    (* One configurator per IPM state (OUT + 4 targets). Writes the
       per-state sName and fDelta. Ticked cyclically in the body AFTER
       fbStates so its writes win over the template baseline
       FB_StateSetup applied via FB_CC_StatePMPSConfig. Idempotent once
       stPositionState.bUpdated trips. *)
    afbStateDefaults : ARRAY[1..5] OF FB_CC_InternalStateConfig[
        (stPositionState := astPositionState[1][E_IPM_States.OUT],
         sName           := 'OUT',
         fDelta          := FDELTA_DEFAULT),
        (stPositionState := astPositionState[1][E_IPM_States.TARGET1],
         sName           := 'TARGET1',
         fDelta          := FDELTA_DEFAULT),
        (stPositionState := astPositionState[1][E_IPM_States.TARGET2],
         sName           := 'TARGET2',
         fDelta          := FDELTA_DEFAULT),
        (stPositionState := astPositionState[1][E_IPM_States.TARGET3],
         sName           := 'TARGET3',
         fDelta          := FDELTA_DEFAULT),
        (stPositionState := astPositionState[1][E_IPM_States.TARGET4],
         sName           := 'TARGET4',
         fDelta          := FDELTA_DEFAULT)
    ];

    {attribute 'pytmc' := 'pv: MMS'}
    fbStates : FB_PositionStatePMPSND(
        aiMotionStage         := aiMotionStage,
        astPositionState      := astPositionState,
        nActiveMotorCount     := 1,
        eEnumSet              := eEnumSet,
        eEnumGet              := eEnumGet,
        bEnableMotion         := bEnableMotion,
        eMotionRequestPolicy  := E_MotionRequestPolicy.INTERRUPT,
        bEnableBeamParams     := bEnableBeamParams,
        bEnablePositionLimits := bEnablePositionLimits,
        bReadDBNow            := bReadDBNow,
        bFileReaderBusy       := bFileReaderBusy,
        bFileReaderError      := bFileReaderError,
        fbFFHWO               := fbFFHWO,
        fbArbiter             := fbArbiter,
        sDeviceName           := sDeviceName,
        sTransitionKey        := sTransitionKey
    );

    i : UINT;

    (* Legacy FB_IPM declared two RTD thermocouples with pytmc PVs
       (RTD:01 / RTD:02) but never called their bodies, so they had
       no runtime effect and exposed no live values to EPICS. Kept
       commented for traceability and to make re-enabling trivial:
       drop the comment, add a cyclic
           fbRTD1();
           fbRTD2();
       below the state-defaults loop, and decide whether to gate them
       with bVeto (e.g. on eEnumGet = E_IPM_States.OUT) per the GBS
       in-beam RTD pattern.

    {attribute 'pytmc' := 'pv: RTD:01'}
    fbRTD1 : FB_CC_TempSensor;

    {attribute 'pytmc' := 'pv: RTD:02'}
    fbRTD2 : FB_CC_TempSensor;
    *)
END_VAR
VAR_OUTPUT
    // The current position state as an enum.
    {attribute 'pytmc' := '
        pv: MMS:STATE:GET
        io: i
    '}
    eEnumGet: E_IPM_States;
    // The PMPS database lookup associated with the current position state.
    stDbStateParams: ST_DbStateParams;
END_VAR
VAR CONSTANT
    (* IPM-wide default tolerance for state in-position detection,
       applied per-state by afbStateDefaults. *)
    FDELTA_DEFAULT : LREAL := 2;
END_VAR

(* Nil-ref guards: every REFERENCE TO backing field must be bound. *)
IF NOT __ISVALIDREF(aiMotionStage)
   OR NOT __ISVALIDREF(astPositionState)
   OR NOT __ISVALIDREF(fbFFHWO)
   OR NOT __ISVALIDREF(fbArbiter) THEN
    RETURN;
END_IF

(* Device-side per-state defaults (afbStateDefaults) are written
   once in FB_CC_InternalStateConfig.CallAfterInit; no cyclic tick. *)
fbStates(stDbStateParams=> stDbStateParams);

(* Auto-fired after FB_Init. fbStates' inline-init ran first and
   forwarded nil refs, so this re-supplies the now-valid refs via
   fbStates.CallAfterInitStateMover / CallAfterInitPMPS and writes the
   per-state device defaults. *)
{attribute 'call_after_init'}
METHOD CallAfterInit
afbStateDefaults[1].CallAfterInit(stPositionState := THIS^.astPositionState[1][E_IPM_States.OUT]);
afbStateDefaults[2].CallAfterInit(stPositionState := THIS^.astPositionState[1][E_IPM_States.TARGET1]);
afbStateDefaults[3].CallAfterInit(stPositionState := THIS^.astPositionState[1][E_IPM_States.TARGET2]);
afbStateDefaults[4].CallAfterInit(stPositionState := THIS^.astPositionState[1][E_IPM_States.TARGET3]);
afbStateDefaults[5].CallAfterInit(stPositionState := THIS^.astPositionState[1][E_IPM_States.TARGET4]);

THIS^.fbStates.CallAfterInitStateMover(
    aiMotionStage         := aiMotionStage,
    astPositionState      := astPositionState,
    nActiveMotorCount     := 1,
    eEnumSet              := eEnumSet,
    eEnumGet              := eEnumGet,
    bEnableMotion         := bEnableMotion,
    eMotionRequestPolicy  := E_MotionRequestPolicy.INTERRUPT,
);

THIS^.fbStates.CallAfterInitPMPS(
    aiMotionStage         := aiMotionStage,
    astPositionState      := astPositionState,
    bEnableBeamParams     := bEnableBeamParams,
    bEnablePositionLimits := bEnablePositionLimits,
    bReadDBNow            := bReadDBNow,
    bFileReaderBusy       := bFileReaderBusy,
    bFileReaderError      := bFileReaderError,
    fbFFHWO               := fbFFHWO,
    fbArbiter             := fbArbiter,
    sDeviceName           := sDeviceName,
    sTransitionKey        := sTransitionKey
);
END_METHOD

(* Stores FB_Init inputs into instance fields; every non-value input is
   REFERENCE TO, REF= bound for the FB lifetime. fbStates inline-init
   captured these params at construction, so this records the same refs
   on THIS^ for body use and live caller writes. *)
{attribute 'analysis' := '-33'}
METHOD FB_Init : BOOL
VAR_INPUT
    bInitRetains           : BOOL;
    bInCopyCode            : BOOL;
    aiMotionStage          : REFERENCE TO ARRAY[1..MotionConstants.MAX_STATE_MOTORS] OF I_MotionStage;
    astPositionState       : REFERENCE TO ARRAY[1..MotionConstants.MAX_STATE_MOTORS]
                                            OF ARRAY[1..GeneralConstants.MAX_STATES] OF ST_PositionState;
    fbFFHWO                : REFERENCE TO FB_HardwareFFOutput;
    fbArbiter              : REFERENCE TO FB_Arbiter;
    sDeviceName            : STRING;
    sTransitionKey         : STRING;
    bEnableBeamParams      : BOOL;
    bEnablePositionLimits  : BOOL;
    bReadDBNow             : BOOL;

    bFileReaderBusy       : REFERENCE TO BOOL;
    bFileReaderError      : REFERENCE TO BOOL;
END_VAR
THIS^.aiMotionStage    REF= aiMotionStage;
THIS^.astPositionState REF= astPositionState;
THIS^.fbFFHWO          REF= fbFFHWO;
THIS^.fbArbiter        REF= fbArbiter;
THIS^.sDeviceName      := sDeviceName;
THIS^.sTransitionKey   := sTransitionKey;
THIS^.bEnableBeamParams     := bEnableBeamParams;
THIS^.bEnablePositionLimits := bEnablePositionLimits;
THIS^.bReadDBNow            := bReadDBNow;
THIS^.bFileReaderBusy       REF= bFileReaderBusy;
THIS^.bFileReaderError      REF= bFileReaderError;
END_METHOD

END_FUNCTION_BLOCK

// ---- Tests/FB_LICTest.TcPOU
FUNCTION_BLOCK FB_LICTest EXTENDS FB_TestSuite
VAR
    (* Caller-owned axis, persistent storage, and Y motor.
       In a real PRG the AxisRef would come from MAIN.Mxx. *)
    axRef    : AXIS_REF;
    fbPDS    : LCLS_Tc_DevAbs.FB_PersistentDataStorage;

    (* FB_LIC is single-axis (nActiveMotorCount := 1), so only slot 1
       holds a real motor. aiMotionStage is sized to
       MotionConstants.MAX_STATE_MOTORS to match FB_LIC.FB_Init's
       fixed-size signature; slots 2-4 default-init to a nil interface
       and are never touched. *)
    fbMotorY : FB_MotionStageNC(AxisRef := axRef, iPersistentDataStorage := fbPDS, sName := 'Y');
    aiMotionStage : ARRAY[1..MotionConstants.MAX_STATE_MOTORS] OF I_MotionStage := [fbMotorY];

    {attribute 'pytmc' := '
        pv: MMS
        array: 1..1 | 1..4
    '}
    astPositionState : ARRAY[1..MotionConstants.MAX_STATE_MOTORS]
                         OF ARRAY[1..GeneralConstants.MAX_STATES] OF ST_PositionState;

    fbFFHWO    : FB_HardwareFFOutput;
    fbArbiter  : FB_Arbiter(1);
    fbSubSysIO : FB_DummyArbIO;

    sDeviceName    : STRING := 'TST:LIC';
    sTransitionKey : STRING := 'TST:LIC-TRANSITION';

    (* Caller-owned file-reader status, bound to FB_LIC by REFERENCE
       TO. In a real PRG these point at MOTION_GVL.fbPmpsFileReader;
       here they stay FALSE so the DB read proceeds. *)
    bFileReaderBusy  : BOOL;
    bFileReaderError : BOOL;

    fbLIC : FB_LIC(
        aiMotionStage         := aiMotionStage,
        astPositionState      := astPositionState,
        fbFFHWO               := fbFFHWO,
        fbArbiter             := fbArbiter,
        sDeviceName           := sDeviceName,
        sTransitionKey        := sTransitionKey,
        bEnableBeamParams     := TRUE,
        bEnablePositionLimits := TRUE,
        bReadDBNow            := TRUE,
        bFileReaderBusy       := bFileReaderBusy,
        bFileReaderError      := bFileReaderError
    );

    (* Per-install PMPS-side state config (caller-owned). Mirrors what
       a real PRG_xxL0_LIC would declare. stDefault is the caller-owned
       baseline template that FB_CC_StatePMPSConfig's inner FB_StateSetup
       preloads from; fbLIC subsequently overrides per-state sName and
       fDelta via its own FB_CC_InternalStateConfig array. *)
    stDefault : ST_PositionState := (
        bMoveOk       := TRUE,
        bValid        := TRUE,
        bUseRawCounts := FALSE
    );

    afbStatePMPS : ARRAY[1..4] OF FB_CC_StatePMPSConfig[
        (stPositionState := astPositionState[1][E_LIC_States.OUT],
         stDefault       := stDefault,
         fPosition       := 10,
         sPmpsState      := 'TST:LIC-OUT'),
        (stPositionState := astPositionState[1][E_LIC_States.MIRROR1],
         stDefault       := stDefault,
         fPosition       := 20,
         sPmpsState      := 'TST:LIC-MIRROR1'),
        (stPositionState := astPositionState[1][E_LIC_States.MIRROR2],
         stDefault       := stDefault,
         fPosition       := 30,
         sPmpsState      := 'TST:LIC-MIRROR2'),
        (stPositionState := astPositionState[1][E_LIC_States.TARGET],
         stDefault       := stDefault,
         fPosition       := 40,
         sPmpsState      := 'TST:LIC-TARGET')
    ];

    bFirstScan : BOOL := TRUE;
    i          : UINT;
END_VAR



TestStateMove();

(*
    Smoke test for LIC state-move wiring. Walks OUT then MIRROR1 and
    asserts each lands within fTolerance of the configured fPosition.
    Mirrors FB_REFTest: stageReady gate up front, NOT bMoving +
    position-tolerance check per state, 60s watchdog, on timeout
    AssertTrue(FALSE, ...) with the current step and observed
    position. Two moves is enough to exercise the FB wiring; the
    motion stack itself is covered by the
    lcls-twincat-motion-abstraction test suite.
*)
METHOD TestStateMove
VAR_INST
    tonTimer  : TON;
    nTestStep : INT := 0;
    fObserved : LREAL;
END_VAR
VAR CONSTANT
    fTolerance : LREAL := 2.0;
END_VAR
TEST('TestLICStateMove');

tonTimer(IN := TRUE, PT := T#60s);
fObserved := fbMotorY.stMotionStatus.fActPosition;

CASE nTestStep OF
    0:
        IF bFirstScan THEN
            fbMotorY.SetModeEnableLimits(
                LimBackward    := TRUE,
                LimForward     := TRUE,
                HomeEnable     := FALSE,
                BrakeMode      := E_StageBrakeMode.IF_ENABLED,
                EnableMode     := E_StageEnableMode.DURING_MOTION,
                HomeMode       := E_EpicsHomeCmd.LOW_LIMIT,
                UserEnable     := TRUE,
                HardwareEnable := TRUE
            );
            fbMotorY.SetVelocity(Velocity := 15.5);
            fbMotorY.RestoreMotionParams      := FALSE;
            fbMotorY.DoNotRestoreNcParameters := TRUE;
            bFileReaderBusy  := TRUE;
            bFileReaderError := FALSE;
            bFirstScan := FALSE;
        END_IF

        IF fbMotorY.stMotionStatus.bStageReady
           AND NOT fbMotorY.stMotionStatus.bError THEN
            fbLIC.eEnumSet := E_LIC_States.OUT;
            nTestStep      := 1;
        END_IF
    1:
        (* OUT is configured at fPosition := 10 in afbStatePMPS[1]. *)
        IF fbLIC.eEnumGet = E_LIC_States.OUT
           AND NOT fbMotorY.stMotionStatus.bMoving
           AND ABS(fObserved - 10.0) <= fTolerance THEN
            fbLIC.eEnumSet := E_LIC_States.MIRROR1;
            nTestStep      := 2;
        END_IF
    2:
        (* MIRROR1 is configured at fPosition := 20 in afbStatePMPS[2]. *)
        IF fbLIC.eEnumGet = E_LIC_States.MIRROR1
           AND NOT fbMotorY.stMotionStatus.bMoving
           AND ABS(fObserved - 20.0) <= fTolerance THEN
            AssertTrue(
                Condition := TRUE,
                Message   := 'TestLICStateMove: OUT then MIRROR1 reached within tolerance');
            nTestStep := 3;
        END_IF
END_CASE


(* Fake PMPS handling. *)
fbSubSysIO(
    LA  := fbArbiter,
    FFO := fbFFHWO
);


fbPDS();
fbMotorY();
fbLIC();

bFileReaderBusy  := FALSE;
bFileReaderError := FALSE;

IF nTestStep = 3 THEN
    TEST_FINISHED();
ELSIF tonTimer.Q THEN
    AssertTrue(
        Condition := FALSE,
        Message   := CONCAT(
            CONCAT(
                CONCAT('TestLICStateMove: timed out at step ', TO_STRING(nTestStep)),
                CONCAT(', eEnumGet=', TO_STRING(TO_UDINT(fbLIC.eEnumGet)))),
            CONCAT(', fActPos=', TO_STRING(fObserved))));
    TEST_FINISHED();
END_IF
END_METHOD

END_FUNCTION_BLOCK

// ---- Devices/LIC/FB_LIC.TcPOU
(* Laser In-Coupling (LIC): thin ND-framework state-mover wrapper.
   Y mover via FB_PositionStatePMPSND (states OUT, MIRROR1, MIRROR2,
   TARGET). Caller-owned motors, stage/state arrays, enum bridge,
   fast-fault and arbiter are injected via FB_Init REFERENCE TO and
   forwarded to fbStates; toggles re-forwarded each cycle. *)
{attribute 'call_after_init'}
FUNCTION_BLOCK FB_LIC
VAR_INPUT
    // Set this to a non-unknown value to request a new move.
    {attribute 'pytmc' := '
        pv: MMS:STATE:SET
        io: io
    '}
    eEnumSet : E_LIC_States;
END_VAR
VAR

    (* REFERENCE TO backing fields populated by FB_Init. Same names as
       FB_Init params; THIS^. disambiguates inside FB_Init.
       Live-bound to caller storage for the lifetime of the FB. *)
    {attribute 'no_copy'}
    aiMotionStage         : REFERENCE TO ARRAY[1..MotionConstants.MAX_STATE_MOTORS] OF I_MotionStage;
    {attribute 'no_copy'}
    astPositionState      : REFERENCE TO ARRAY[1..MotionConstants.MAX_STATE_MOTORS]
                                            OF ARRAY[1..GeneralConstants.MAX_STATES] OF ST_PositionState;
    {attribute 'no_copy'}
    fbFFHWO               : REFERENCE TO FB_HardwareFFOutput;
    {attribute 'no_copy'}
    fbArbiter             : REFERENCE TO FB_Arbiter;
    sDeviceName           : STRING;
    sTransitionKey        : STRING;
    bEnableMotion         : BOOL := TRUE;
    bEnableBeamParams     : BOOL;
    bEnablePositionLimits : BOOL;
    bReadDBNow            : BOOL;

    bFileReaderBusy       : REFERENCE TO BOOL;
    bFileReaderError      : REFERENCE TO BOOL;

    (* One configurator per LIC state (OUT, MIRROR1, MIRROR2, TARGET).
       Writes the per-state sName and fDelta. Ticked cyclically in the
       body AFTER fbStates so its writes win over the template baseline
       FB_StateSetup applied via FB_CC_StatePMPSConfig. Idempotent once
       stPositionState.bUpdated trips. *)
    afbStateDefaults : ARRAY[1..4] OF FB_CC_InternalStateConfig[
        (stPositionState := astPositionState[1][E_LIC_States.OUT],
         sName           := 'OUT',
         fDelta          := FDELTA_DEFAULT),
        (stPositionState := astPositionState[1][E_LIC_States.MIRROR1],
         sName           := 'MIRROR1',
         fDelta          := FDELTA_DEFAULT),
        (stPositionState := astPositionState[1][E_LIC_States.MIRROR2],
         sName           := 'MIRROR2',
         fDelta          := FDELTA_DEFAULT),
        (stPositionState := astPositionState[1][E_LIC_States.TARGET],
         sName           := 'TARGET',
         fDelta          := FDELTA_DEFAULT)
    ];

    {attribute 'pytmc' := 'pv: MMS'}
    fbStates : FB_PositionStatePMPSND(
        aiMotionStage         := aiMotionStage,
        astPositionState      := astPositionState,
        nActiveMotorCount     := 1,
        eEnumSet              := eEnumSet,
        eEnumGet              := eEnumGet,
        bEnableMotion         := bEnableMotion,
        eMotionRequestPolicy  := E_MotionRequestPolicy.INTERRUPT,
        bEnableBeamParams     := bEnableBeamParams,
        bEnablePositionLimits := bEnablePositionLimits,
        bReadDBNow            := bReadDBNow,
        bFileReaderBusy       := bFileReaderBusy,
        bFileReaderError      := bFileReaderError,
        fbFFHWO               := fbFFHWO,
        fbArbiter             := fbArbiter,
        sDeviceName           := sDeviceName,
        sTransitionKey        := sTransitionKey
    );
    i : UINT;
END_VAR
VAR_OUTPUT
    // The current position state as an enum.
    {attribute 'pytmc' := '
        pv: MMS:STATE:GET
        io: i
    '}
    eEnumGet: E_LIC_States;
    // The PMPS database lookup associated with the current position state.
    stDbStateParams: ST_DbStateParams;
END_VAR
VAR CONSTANT
    (* LIC-wide default tolerance for state in-position detection,
       applied per-state by afbStateDefaults. *)
    FDELTA_DEFAULT : LREAL := 2;
END_VAR

(* Nil-ref guards: every REFERENCE TO backing field must be bound. *)
IF NOT __ISVALIDREF(aiMotionStage)
   OR NOT __ISVALIDREF(astPositionState)
   OR NOT __ISVALIDREF(fbFFHWO)
   OR NOT __ISVALIDREF(fbArbiter) THEN
    RETURN;
END_IF

(* Device-side per-state defaults (afbStateDefaults) are written
   once in FB_CC_InternalStateConfig.CallAfterInit; no cyclic tick. *)
fbStates(stDbStateParams=> stDbStateParams);

(* Auto-fired after FB_Init. fbStates' inline-init ran first and
   forwarded nil refs, so this re-supplies the now-valid refs via
   fbStates.CallAfterInitStateMover / CallAfterInitPMPS and writes the
   per-state device defaults. *)
{attribute 'call_after_init'}
METHOD CallAfterInit
afbStateDefaults[1].CallAfterInit(stPositionState := THIS^.astPositionState[1][E_LIC_States.OUT]);
afbStateDefaults[2].CallAfterInit(stPositionState := THIS^.astPositionState[1][E_LIC_States.MIRROR1]);
afbStateDefaults[3].CallAfterInit(stPositionState := THIS^.astPositionState[1][E_LIC_States.MIRROR2]);
afbStateDefaults[4].CallAfterInit(stPositionState := THIS^.astPositionState[1][E_LIC_States.TARGET]);

THIS^.fbStates.CallAfterInitStateMover(
    aiMotionStage         := aiMotionStage,
    astPositionState      := astPositionState,
    nActiveMotorCount     := 1,
    eEnumSet              := eEnumSet,
    eEnumGet              := eEnumGet,
    bEnableMotion         := bEnableMotion,
    eMotionRequestPolicy  := E_MotionRequestPolicy.INTERRUPT,
);

THIS^.fbStates.CallAfterInitPMPS(
    aiMotionStage         := aiMotionStage,
    astPositionState      := astPositionState,
    bEnableBeamParams     := bEnableBeamParams,
    bEnablePositionLimits := bEnablePositionLimits,
    bReadDBNow            := bReadDBNow,
    bFileReaderBusy       := bFileReaderBusy,
    bFileReaderError      := bFileReaderError,
    fbFFHWO               := fbFFHWO,
    fbArbiter             := fbArbiter,
    sDeviceName           := sDeviceName,
    sTransitionKey        := sTransitionKey
);
END_METHOD

(* Stores FB_Init inputs into instance fields; every non-value input is
   REFERENCE TO, REF= bound for the FB lifetime. fbStates inline-init
   captured these params at construction, so this records the same refs
   on THIS^ for body use and live caller writes. *)
{attribute 'analysis' := '-33'}
METHOD FB_Init : BOOL
VAR_INPUT
    bInitRetains           : BOOL;
    bInCopyCode            : BOOL;
    aiMotionStage          : REFERENCE TO ARRAY[1..MotionConstants.MAX_STATE_MOTORS] OF I_MotionStage;
    astPositionState       : REFERENCE TO ARRAY[1..MotionConstants.MAX_STATE_MOTORS]
                                            OF ARRAY[1..GeneralConstants.MAX_STATES] OF ST_PositionState;
    fbFFHWO                : REFERENCE TO FB_HardwareFFOutput;
    fbArbiter              : REFERENCE TO FB_Arbiter;
    sDeviceName            : STRING;
    sTransitionKey         : STRING;
    bEnableBeamParams      : BOOL;
    bEnablePositionLimits  : BOOL;
    bReadDBNow             : BOOL;
    bFileReaderBusy       : REFERENCE TO BOOL;
    bFileReaderError      : REFERENCE TO BOOL;
END_VAR
THIS^.aiMotionStage    REF= aiMotionStage;
THIS^.astPositionState REF= astPositionState;
THIS^.fbFFHWO          REF= fbFFHWO;
THIS^.fbArbiter        REF= fbArbiter;
THIS^.sDeviceName      := sDeviceName;
THIS^.sTransitionKey   := sTransitionKey;
THIS^.bEnableBeamParams     := bEnableBeamParams;
THIS^.bEnablePositionLimits := bEnablePositionLimits;
THIS^.bReadDBNow            := bReadDBNow;
THIS^.bFileReaderBusy       REF= bFileReaderBusy;
THIS^.bFileReaderError      REF= bFileReaderError;
END_METHOD

END_FUNCTION_BLOCK

// ---- Tests/FB_PPMTest.TcPOU
FUNCTION_BLOCK FB_PPMTest EXTENDS FB_TestSuite
VAR
    (* Caller-owned axis, persistent storage, and Y motor.
       In a real PRG the AxisRef would come from MAIN.Mxx. *)
    axRef    : AXIS_REF;
    fbPDS    : LCLS_Tc_DevAbs.FB_PersistentDataStorage;

    (* FB_PPM is single-axis (nActiveMotorCount := 1), so only slot 1
       holds a real motor. aiMotionStage is sized to
       MotionConstants.MAX_STATE_MOTORS to match FB_PPM.FB_Init's
       fixed-size signature; slots 2-4 default-init to a nil interface
       and are never touched. *)
    fbMotorY : FB_MotionStageNC(AxisRef := axRef, iPersistentDataStorage := fbPDS, sName := 'Y');
    aiMotionStage : ARRAY[1..MotionConstants.MAX_STATE_MOTORS] OF I_MotionStage := [fbMotorY];

    {attribute 'pytmc' := '
        pv: MMS
        array: 1..1 | 1..4
    '}
    astPositionState : ARRAY[1..MotionConstants.MAX_STATE_MOTORS]
                         OF ARRAY[1..GeneralConstants.MAX_STATES] OF ST_PositionState;

    fbFFHWO    : FB_HardwareFFOutput;
    fbArbiter  : FB_Arbiter(1);
    fbSubSysIO : FB_DummyArbIO;

    sDeviceName    : STRING := 'TST:PPM';
    sTransitionKey : STRING := 'TST:PPM-TRANSITION';

    (* Caller-owned file-reader status, bound to FB_PPM by REFERENCE
       TO. In a real PRG these point at MOTION_GVL.fbPmpsFileReader;
       here they stay FALSE so the DB read proceeds. *)
    bFileReaderBusy  : BOOL;
    bFileReaderError : BOOL;

    fbPPM : FB_PPM(
        aiMotionStage         := aiMotionStage,
        astPositionState      := astPositionState,
        fbFFHWO               := fbFFHWO,
        fbArbiter             := fbArbiter,
        sDeviceName           := sDeviceName,
        sTransitionKey        := sTransitionKey,
        bEnableBeamParams     := TRUE,
        bEnablePositionLimits := TRUE,
        bReadDBNow            := TRUE,
        bFileReaderBusy       := bFileReaderBusy,
        bFileReaderError      := bFileReaderError
    );

    (* Per-install PMPS-side state config (caller-owned). Mirrors what
       a real PRG_xxL0_PPM would declare. stDefault is the caller-owned
       baseline template that FB_CC_StatePMPSConfig's inner FB_StateSetup
       preloads from; fbPPM subsequently overrides per-state sName and
       fDelta via its own FB_CC_InternalStateConfig array. *)
    stDefault : ST_PositionState := (
        bMoveOk       := TRUE,
        bValid        := TRUE,
        bUseRawCounts := FALSE
    );

    afbStatePMPS : ARRAY[1..4] OF FB_CC_StatePMPSConfig[
        (stPositionState := astPositionState[1][E_PPM_States.OUT],
         stDefault       := stDefault,
         fPosition       := 10,
         sPmpsState      := 'TST:PPM-OUT'),
        (stPositionState := astPositionState[1][E_PPM_States.POWERMETER],
         stDefault       := stDefault,
         fPosition       := 20,
         sPmpsState      := 'TST:PPM-POWERMETER'),
        (stPositionState := astPositionState[1][E_PPM_States.YAG1],
         stDefault       := stDefault,
         fPosition       := 30,
         sPmpsState      := 'TST:PPM-YAG1'),
        (stPositionState := astPositionState[1][E_PPM_States.YAG2],
         stDefault       := stDefault,
         fPosition       := 40,
         sPmpsState      := 'TST:PPM-YAG2')
    ];

    bFirstScan : BOOL := TRUE;
    i          : UINT;
END_VAR

TestStateMove();
TestTempFFO();

METHOD AssertBothTempFault
VAR_INPUT
    Message : STRING;
END_VAR
AssertFalse(
    fbPPM.fbYagTempSensor.FFO.i_xOK,
    CONCAT('PPM yag temp sensor expected fault: ', Message)
);
AssertFalse(
    fbPPM.fbPowerMeter.fbTempSensor.FFO.i_xOK,
    CONCAT('PPM pm temp sensor expected fault: ', Message)
);
END_METHOD

METHOD AssertNeitherTempFault
VAR_INPUT
    Message : STRING;
END_VAR
AssertTrue(
    fbPPM.fbYagTempSensor.FFO.i_xOK,
    CONCAT('PPM yag temp sensor expected ok: ', Message)
);
AssertTrue(
    fbPPM.fbPowerMeter.fbTempSensor.FFO.i_xOK,
    CONCAT('PPM pm temp sensor expected ok: ', Message)
);
END_METHOD

METHOD SetPPMTemp
VAR_INPUT
    iTempC : INT;
END_VAR
VAR
    ptr : POINTER TO INT;
END_VAR
ptr  := ADR(fbPPM.fbYagTempSensor.iRaw);
ptr^ := iTempC * 10;

ptr  := ADR(fbPPM.fbPowerMeter.fbTempSensor.iRaw);
ptr^ := iTempC * 10;
END_METHOD

(*
    Smoke test for PPM state-move wiring. Walks OUT then POWERMETER
    and asserts each lands within fTolerance of the configured
    fPosition. Mirrors FB_REFTest: stageReady gate up front, NOT
    bMoving + position-tolerance check per state, 60s watchdog, on
    timeout AssertTrue(FALSE, ...) with the current step and observed
    position. Two moves is enough to exercise the FB wiring; the
    motion stack itself is covered by the
    lcls-twincat-motion-abstraction test suite.
*)
METHOD TestStateMove
VAR_INST
    tonTimer  : TON;
    nTestStep : INT := 0;
    fObserved : LREAL;
END_VAR
VAR CONSTANT
    fTolerance : LREAL := 2.0;
END_VAR
TEST('TestPPMStateMove');

tonTimer(IN := TRUE, PT := T#60s);
fObserved := fbMotorY.stMotionStatus.fActPosition;

CASE nTestStep OF
    0:
        IF bFirstScan THEN
            fbMotorY.SetModeEnableLimits(
                LimBackward    := TRUE,
                LimForward     := TRUE,
                HomeEnable     := FALSE,
                BrakeMode      := E_StageBrakeMode.IF_ENABLED,
                EnableMode     := E_StageEnableMode.DURING_MOTION,
                HomeMode       := E_EpicsHomeCmd.LOW_LIMIT,
                UserEnable     := TRUE,
                HardwareEnable := TRUE
            );
            fbMotorY.SetVelocity(Velocity := 15.5);
            fbMotorY.RestoreMotionParams      := FALSE;
            fbMotorY.DoNotRestoreNcParameters := TRUE;
            bFileReaderBusy  := TRUE;
            bFileReaderError := FALSE;
            bFirstScan := FALSE;
        END_IF
        nTestStep      := 1;
    1:
        IF fbMotorY.stMotionStatus.bStageReady
           AND NOT fbMotorY.stMotionStatus.bError THEN
            fbPPM.eEnumSet := E_PPM_States.OUT;
            nTestStep      := 2;
        END_IF
    2:
        (* OUT is configured at fPosition := 10 in afbStatePMPS[1]. *)
        IF fbPPM.eEnumGet = E_PPM_States.OUT
           AND NOT fbMotorY.stMotionStatus.bMoving
           AND ABS(fObserved - 10.0) <= fTolerance THEN
            fbPPM.eEnumSet := E_PPM_States.POWERMETER;
            nTestStep      := 3;
        END_IF
    3:
        (* POWERMETER is configured at fPosition := 20 in afbStatePMPS[2]. *)
        IF fbPPM.eEnumGet = E_PPM_States.POWERMETER
           AND NOT fbMotorY.stMotionStatus.bMoving
           AND ABS(fObserved - 20.0) <= fTolerance THEN
            AssertTrue(
                Condition := TRUE,
                Message   := 'TestPPMStateMove: OUT then POWERMETER reached within tolerance');
            nTestStep := 4;
        END_IF
END_CASE

(* Fake PMPS handling. *)
fbSubSysIO(
    LA  := fbArbiter,
    FFO := fbFFHWO
);

fbPDS();
fbMotorY();
fbPPM();


bFileReaderBusy  := FALSE;
bFileReaderError := FALSE;

IF nTestStep = 4 THEN
    TEST_FINISHED();
ELSIF tonTimer.Q THEN
    AssertTrue(
        Condition := FALSE,
        Message   := CONCAT(
            CONCAT(
                CONCAT('TestPPMStateMove: timed out at step ', TO_STRING(nTestStep)),
                CONCAT(', eEnumGet=', TO_STRING(TO_UDINT(fbPPM.eEnumGet)))),
            CONCAT(', fActPos=', TO_STRING(fObserved))));
    TEST_FINISHED();
END_IF
END_METHOD

METHOD TestTempFFO
VAR_INST
    tonTimer    : TON;
    nStep       : UINT := 0;
    bOutChecked : BOOL := FALSE;
    bInChecked  : BOOL := FALSE;
END_VAR
VAR CONSTANT
    nLastStep : UINT := 3;
END_VAR

(* Do we fault at the correct times?
   Parasitically depends on state move test. *)
TEST('TestPPMTempFFO');

(* Prepare a timeout *)
tonTimer(IN := TRUE, PT := T#10s);

CASE nStep OF
    0:
        (* Set the thermocouple temperatures to crazy high number. *)
        SetPPMTemp(100);
        nStep := nStep + 1;
    1:
        (* Wait till we see "OUT" state and one other state (OUT
           should be no fault). *)
        IF fbPPM.eEnumGet = E_PPM_States.OUT THEN
            AssertNeitherTempFault('was in out position');
            bOutChecked := TRUE;
        ELSIF fbPPM.eEnumGet <> E_PPM_States.Unknown THEN
            AssertBothTempFault('was in a target position');
            bInChecked := TRUE;
        END_IF
        IF bOutChecked AND bInChecked THEN
            nStep := nStep + 1;
        END_IF
    2:
        (* Set the thermocouple temperatures to low again. *)
        SetPPMTemp(0);
        nStep := nStep + 1;
    3:
        AssertNeitherTempFault('has low temp reading');
        nStep := nStep + 1;
END_CASE

IF tonTimer.Q OR nStep > nLastStep THEN
    AssertFalse(tonTimer.Q, 'Timeout in PPM temp FFO test');
    TEST_FINISHED();
END_IF
END_METHOD

END_FUNCTION_BLOCK

// ---- Devices/PPM/FB_PPM.TcPOU
(* Power and Profile Monitor (PPM): thin ND-framework state-mover wrapper.
   Y mover via FB_PositionStatePMPSND (states OUT, POWERMETER, YAG1, YAG2),
   plus a tick site for power meter, GigE camera/illuminator, flow meter,
   YAG thermocouple and flow switch. Caller-owned deps injected via FB_Init
   REFERENCE TO and forwarded to fbStates; toggles re-forwarded each cycle. *)
{attribute 'call_after_init'}
FUNCTION_BLOCK FB_PPM
VAR_INPUT
    // Set this to a non-unknown value to request a new move.
    {attribute 'pytmc' := '
        pv: MMS:STATE:SET
        io: io
    '}
    eEnumSet : E_PPM_States;
    (* Flow meter offset in engineering units (per-install). *)
    fFlowOffset   : LREAL := 0;
    (* Power-meter responsivity (calibrated per gentec); if zero the
       responsive energy is not calculated. *)
    fResponsivity : LREAL;

    (* Passed straight through to FB_PPM_PowerMeter's analog input.
       Defaults are correct for EL3062; EL3602 needs iTermBits:=31
       with fTermMax/fTermMin matching the terminal's configured
       voltage range. *)
    iTermBits : UINT := 15;
    fTermMax  : REAL := 10000;
    fTermMin  : REAL := 0;

END_VAR
VAR
    {attribute 'pytmc' := 'pv: SPM'}
    fbPowerMeter : FB_PPM_PowerMeter;

    {attribute 'pytmc' := 'pv: CAM'}
    fbGige : FB_PPM_Gige;

    {attribute 'pytmc' := 'pv: FWM'}
    fbFlowMeter : FB_AnalogInput := (iTermBits := 15, fTermMax := 60, fTermMin := 0);

    {attribute 'pytmc' := 'pv: YAG:STC'}
    fbYagTempSensor : FB_CC_TempSensor;

    {attribute 'pytmc' := 'pv: FSW'}
    fbFlowSwitch : FB_XTES_Flowswitch;

    (* REFERENCE TO backing fields populated by FB_Init. Same names as
       FB_Init params; THIS^. disambiguates inside FB_Init.
       Live-bound to caller storage for the lifetime of the FB. *)
    {attribute 'no_copy'}
    aiMotionStage         : REFERENCE TO ARRAY[1..MotionConstants.MAX_STATE_MOTORS] OF I_MotionStage;
    {attribute 'no_copy'}
    astPositionState      : REFERENCE TO ARRAY[1..MotionConstants.MAX_STATE_MOTORS]
                                            OF ARRAY[1..GeneralConstants.MAX_STATES] OF ST_PositionState;
    {attribute 'no_copy'}
    fbFFHWO               : REFERENCE TO FB_HardwareFFOutput;
    {attribute 'no_copy'}
    fbArbiter             : REFERENCE TO FB_Arbiter;
    sDeviceName           : STRING;
    sTransitionKey        : STRING;
    bEnableMotion         : BOOL := TRUE;
    bEnableBeamParams     : BOOL;
    bEnablePositionLimits : BOOL;
    bReadDBNow            : BOOL;

    bFileReaderBusy       : REFERENCE TO BOOL;
    bFileReaderError      : REFERENCE TO BOOL;

    (* One configurator per PPM state. Writes the per-state sName and
       fDelta. Ticked cyclically in the body AFTER fbStates so its
       writes win over the template baseline FB_StateSetup applied via
       FB_CC_StatePMPSConfig. Idempotent once stPositionState.bUpdated
       trips. *)
    afbStateDefaults : ARRAY[1..4] OF FB_CC_InternalStateConfig[
        (stPositionState := astPositionState[1][E_PPM_States.OUT],
         sName           := 'OUT',
         fDelta          := FDELTA_DEFAULT),
        (stPositionState := astPositionState[1][E_PPM_States.POWERMETER],
         sName           := 'POWERMETER',
         fDelta          := FDELTA_DEFAULT),
        (stPositionState := astPositionState[1][E_PPM_States.YAG1],
         sName           := 'YAG1',
         fDelta          := FDELTA_DEFAULT),
        (stPositionState := astPositionState[1][E_PPM_States.YAG2],
         sName           := 'YAG2',
         fDelta          := FDELTA_DEFAULT)
    ];

    {attribute 'pytmc' := 'pv: MMS'}
    fbStates : FB_PositionStatePMPSND(
        aiMotionStage         := aiMotionStage,
        astPositionState      := astPositionState,
        nActiveMotorCount     := 1,
        eEnumSet              := eEnumSet,
        eEnumGet              := eEnumGet,
        bEnableMotion         := bEnableMotion,
        eMotionRequestPolicy  := E_MotionRequestPolicy.INTERRUPT,
        bEnableBeamParams     := bEnableBeamParams,
        bEnablePositionLimits := bEnablePositionLimits,
        bReadDBNow            := bReadDBNow,
        bFileReaderBusy       := bFileReaderBusy,
        bFileReaderError      := bFileReaderError,
        fbFFHWO               := fbFFHWO,
        fbArbiter             := fbArbiter,
        sDeviceName           := sDeviceName,
        sTransitionKey        := sTransitionKey
    );

    i : UINT;
END_VAR

VAR_OUTPUT
    // The current position state as an enum.
    {attribute 'pytmc' := '
        pv: MMS:STATE:GET
        io: i
    '}
    eEnumGet: E_PPM_States;
    // The PMPS database lookup associated with the current position state.
    stDbStateParams: ST_DbStateParams;
END_VAR

VAR CONSTANT
    (* PPM-wide default tolerance for state in-position detection,
       applied per-state by afbStateDefaults. *)
    FDELTA_DEFAULT : LREAL := 2;
END_VAR

(* Nil-ref guards: every REFERENCE TO backing field must be bound. *)
IF NOT __ISVALIDREF(aiMotionStage)
   OR NOT __ISVALIDREF(astPositionState)
   OR NOT __ISVALIDREF(fbFFHWO)
   OR NOT __ISVALIDREF(fbArbiter) THEN
    RETURN;
END_IF

(* Device-side per-state defaults (afbStateDefaults) are written
   once in FB_CC_InternalStateConfig.CallAfterInit; no cyclic tick. *)
fbStates(stDbStateParams=> stDbStateParams);

(* Power meter: consumes the current state enum + axis NC state for
   background auto-collection, and the PMPS DB temp setpoint to drive
   its thermocouple FFO. Vetoes the temp FFO outside POWERMETER. *)
fbPowerMeter(
    fTempSP       := fbStates.stDbStateParams.stReactiveParams.nTempSP,
    bVetoTempFFO  := eEnumGet <> E_PPM_States.POWERMETER,
    sDeviceName   := sDeviceName,
    fbFFHWO       := fbFFHWO,
    eEnumGet      := eEnumGet,
    stYAxisState  := aiMotionStage[1].Axis.NcToPlc.AxisState,
    fResponsivity := fResponsivity,
    iTermBits     := iTermBits,
    fTermMax      := fTermMax,
    fTermMin      := fTermMin
);

fbGige();
fbFlowMeter(fOffset := fFlowOffset);

(* YAG thermocouple: only faults when the YAG is actually in-beam
   (i.e. not OUT). Driven by the same PMPS DB temp setpoint. *)
fbYagTempSensor(
    fFaultThreshold := fbStates.stDbStateParams.stReactiveParams.nTempSP,
    bVeto           := eEnumGet = E_PPM_States.OUT,
    sDevName        := sDeviceName,
    io_fbFFHWO      := fbFFHWO
);

fbFlowSwitch();

(* Auto-fired after FB_Init. fbStates' inline-init ran first and
   forwarded nil refs, so this re-supplies the now-valid refs via
   fbStates.CallAfterInitStateMover / CallAfterInitPMPS and writes the
   per-state device defaults. *)
{attribute 'call_after_init'}
METHOD CallAfterInit
afbStateDefaults[1].CallAfterInit(stPositionState := THIS^.astPositionState[1][E_PPM_States.OUT]);
afbStateDefaults[2].CallAfterInit(stPositionState := THIS^.astPositionState[1][E_PPM_States.POWERMETER]);
afbStateDefaults[3].CallAfterInit(stPositionState := THIS^.astPositionState[1][E_PPM_States.YAG1]);
afbStateDefaults[4].CallAfterInit(stPositionState := THIS^.astPositionState[1][E_PPM_States.YAG2]);

THIS^.fbStates.CallAfterInitStateMover(
    aiMotionStage         := aiMotionStage,
    astPositionState      := astPositionState,
    nActiveMotorCount     := 1,
    eEnumSet              := eEnumSet,
    eEnumGet              := eEnumGet,
    bEnableMotion         := bEnableMotion,
    eMotionRequestPolicy  := E_MotionRequestPolicy.INTERRUPT,
);

THIS^.fbStates.CallAfterInitPMPS(
    aiMotionStage         := aiMotionStage,
    astPositionState      := astPositionState,
    bEnableBeamParams     := bEnableBeamParams,
    bEnablePositionLimits := bEnablePositionLimits,
    bReadDBNow            := bReadDBNow,
    bFileReaderBusy       := bFileReaderBusy,
    bFileReaderError      := bFileReaderError,
    fbFFHWO               := fbFFHWO,
    fbArbiter             := fbArbiter,
    sDeviceName           := sDeviceName,
    sTransitionKey        := sTransitionKey
);
END_METHOD

(* Stores FB_Init inputs into instance fields; every non-value input is
   REFERENCE TO, REF= bound for the FB lifetime. fbStates inline-init
   captured these params at construction, so this records the same refs
   on THIS^ for body use and live caller writes. *)
{attribute 'analysis' := '-33'}
METHOD FB_Init : BOOL
VAR_INPUT
    bInitRetains           : BOOL;
    bInCopyCode            : BOOL;
    aiMotionStage          : REFERENCE TO ARRAY[1..MotionConstants.MAX_STATE_MOTORS] OF I_MotionStage;
    astPositionState       : REFERENCE TO ARRAY[1..MotionConstants.MAX_STATE_MOTORS]
                                            OF ARRAY[1..GeneralConstants.MAX_STATES] OF ST_PositionState;
    fbFFHWO                : REFERENCE TO FB_HardwareFFOutput;
    fbArbiter              : REFERENCE TO FB_Arbiter;
    sDeviceName            : STRING;
    sTransitionKey         : STRING;
    bEnableBeamParams      : BOOL;
    bEnablePositionLimits  : BOOL;
    bReadDBNow             : BOOL;
    bFileReaderBusy       : REFERENCE TO BOOL;
    bFileReaderError      : REFERENCE TO BOOL;
END_VAR
THIS^.aiMotionStage    REF= aiMotionStage;
THIS^.astPositionState REF= astPositionState;
THIS^.fbFFHWO          REF= fbFFHWO;
THIS^.fbArbiter        REF= fbArbiter;
THIS^.sDeviceName      := sDeviceName;
THIS^.sTransitionKey   := sTransitionKey;
THIS^.bEnableBeamParams     := bEnableBeamParams;
THIS^.bEnablePositionLimits := bEnablePositionLimits;
THIS^.bReadDBNow            := bReadDBNow;
THIS^.bFileReaderBusy       REF= bFileReaderBusy;
THIS^.bFileReaderError      REF= bFileReaderError;
END_METHOD

END_FUNCTION_BLOCK

// ---- Devices/PPM/FB_PPM_PowerMeter.TcPOU
FUNCTION_BLOCK FB_PPM_PowerMeter
VAR_INPUT
    fTempSP: REAL;
    bVetoTempFFO: BOOL;
    sDeviceName: STRING;

    // Used to know when to stop background auto-collection
    eEnumGet: E_PPM_States;
    stYAxisState: DWORD;

    // Calibrated for each gentec, should be passed as input
    // If not set, responsive energy will not be calculated
    {attribute 'pytmc' := '
        pv: RESP
        io: i
        field: EGU V/W
    '}
    fResponsivity: LREAL;

    // Passed to FB_AnalogInput
    // The initial values are correct for EL3062,
    // but not for EL3602, which needs iTermBits:=31
    // with fTermMax and fTermMin dependent on what
    // range the terminal was configured to use
    // (default -10000mV to +10000mV)
    iTermBits : UINT := 15;
    fTermMax : REAL := 10000;
    fTermMin: REAL := 0;
END_VAR
VAR_IN_OUT
    fbFFHWO: FB_HardwareFFOutput;
END_VAR
VAR
    iVoltageINT AT %I*: DINT;

    {attribute 'pytmc' := '
        pv: VOLT
        io: input
        field: EGU mV
    '}
    fVoltage: LREAL;

    {attribute 'pytmc' := '
        pv: VOLT_BUFFER
        io: input
        field: EGU mV
    '}
    fVoltageBuffer: ARRAY[1..1000] OF LREAL;

    {attribute 'pytmc' := '
        pv: STC
        io: input
    '}
    fbTempSensor: FB_CC_TempSensor;


    fFrequency: REAL;
    // Used to get beam rate
    {attribute 'pytmc' := '
        pv: SXR_NC_BeamRateFromEpics
        link: EVNT:SYS0:1:NC_SOFTRATE
    '}
    fSXR_NC_Frequency: REAL;
    {attribute 'pytmc' := '
        pv: SXR_SC_BeamRateFromEpics
        link: TPG:SYS0:1:DST04:RATE_RBV
    '}
    uSXR_SC_Frequency: UINT;

    {attribute 'pytmc' := '
        pv: HXR_NC_BeamRateFromEpics
        link: EVNT:SYS0:1:NC_HARDRATE
    '}
    fHXR_NC_Frequency: REAL;
    {attribute 'pytmc' := '
        pv: HXR_SC_BeamRateFromEpics
        link: TPG:SYS0:1:DST03:RATE_RBV
    '}
    uHXR_SC_Frequency: UINT;

    // Pulse-by-pulse energy and buffer
    {attribute 'pytmc' := '
        pv: MJ
        io: i
        field: EGU mJ
    '}
    fCalibMJ: LREAL;
    {attribute 'pytmc' := '
        pv: MJ_BUFFER
        io: i
        field: EGU mJ
    '}
    fCalibMJBuffer: ARRAY[1..1000] OF LREAL;

    // Wattage and buffer
    {attribute 'pytmc' := '
        pv: WATT
        io: i
        field: EGU mW
    '}
    fPulseWattage: LREAL;
    {attribute 'pytmc' := '
        pv: WATT_BUFFER
        io: i
        field: EGU mW
    '}
    fPulseWattageBuffer: ARRAY[1..1000] OF LREAL;

    // Background voltage
    {attribute 'pytmc' := '
        pv: BACK:VOLT
        io: io
        field: EGU mV
    '}
    fBackgroundVoltage: LREAL;

    // Internal variables for background voltage auto-collection
    fBackgroundVoltageAcc: LREAL;
    uAccCount: UINT;
    fBackgroundVoltageSum: LREAL;
    fBackgroundVoltageStale: LREAL;
    tonBackgroundAutoCollecting: TON;
    fBackgroundVoltageBuffer: ARRAY[1..100] OF LREAL;
    udBackgroundVoltageBufferIndex: UDINT := 1;
    rTrig_Background : R_TRIG;
    i: UDINT;
    // Used to reset auto-collected background buffer, and fBackgroundVoltage if in Auto mode
    {attribute 'pytmc' := '
        pv: BACK:RESET
        io: io
    '}
    bResetAutoBackground: BOOL;

    // In manual mode, auto-background updates buffer but does not change fBackgroundVoltage
    {attribute 'pytmc' := '
        pv: BACK:MODE
        io: io
    '}
    BACKGROUND_MODE: (Manual, Auto) := Auto;

    // Boolean to trigger collection of background voltages
    {attribute 'pytmc' := '
        pv: BACK:COLL
        io: io
    '}
    bBackgroundCollect: BOOL;

    // Time in seconds to collect background voltages for
    {attribute 'pytmc' := '
        pv: BACK:TIME
        io: io
        field: EGU s
    '}
    uBackgroundCollectionTime: UINT := 60;
    tofBackgroundCollecting: TOF;
    udBackgroundManualCount: UDINT;
    // Boolean indicating when background is being manually collected
    {attribute 'pytmc' := '
        pv: BACK:MANUAL_COLLECTING
        io: i
    '}
    bBackgroundCollecting: BOOL := FALSE;

    fbGetPMVoltage: FB_AnalogInput;

    fbVoltageBuffer: FB_LREALBuffer;
    fbPulseWattageBuffer: FB_LREALBuffer;
    fbCalibMJBuffer: FB_LREALBuffer;
END_VAR

fbTempSensor(
    fFaultThreshold:=fTempSP,
    bVeto:=bVetoTempFFO,
    sDevName:=sDeviceName,
    io_fbFFHWO:=fbFFHWO,
);

// Convert the terminal's integer into a value in millivolts
// If you get a compile-time error about converting type DINT
// to type INT, update your lcls-general version to at least
// v2.12.0
fbGetPMVoltage(
    iRaw := iVoltageINT,
    iTermBits := iTermBits,
    fTermMax := fTermMax,
    fTermMin := fTermMin,
    fReal => fVoltage);

rTrig_Background(CLK:=(eEnumGet <> E_PPM_States.OUT OR stYAxisState <> 0));
// Reset buffer and related variables
IF rTrig_Background.Q OR bResetAutoBackground THEN
    IF bResetAutoBackground THEN
        bResetAutoBackground := FALSE;
        IF BACKGROUND_MODE = Auto THEN
            fBackgroundVoltage := 0;
        END_IF
    ELSE
        // Dump 5s worth of readings
        IF udBackgroundVoltageBufferIndex > 6 THEN
            FOR i := (udBackgroundVoltageBufferIndex - 5) TO (udBackgroundVoltageBufferIndex - 1) DO
                fBackgroundVoltageSum := fBackgroundVoltageSum - fBackgroundVoltageBuffer[((i-1) MOD 100) + 1];
            END_FOR
            udBackgroundVoltageBufferIndex := udBackgroundVoltageBufferIndex - 5;
            IF udBackgroundVoltageBufferIndex <> 1 AND BACKGROUND_MODE = Auto THEN
                fBackgroundVoltage := fBackgroundVoltageSum / MIN((udBackgroundVoltageBufferIndex - 1), 100);
            END_IF
        ELSIF BACKGROUND_MODE = Auto THEN
                fBackgroundVoltage := 0;
        END_IF
    END_IF
    fBackgroundVoltageAcc := 0;
    fBackgroundVoltageSum := 0;
    tonBackgroundAutoCollecting(IN := FALSE);
    udBackgroundVoltageBufferIndex := 1;
ELSIF eEnumGet = E_PPM_States.OUT AND stYAxisState = 0 THEN
    tonBackgroundAutoCollecting( IN := TRUE, PT := T#1000MS);
    // Every second, move fBackgroundVoltageAcc into buffer and sum
    IF tonBackgroundAutoCollecting.Q = TRUE THEN
        tonBackgroundAutoCollecting( IN := FALSE);
        fBackgroundVoltageStale := fBackgroundVoltageBuffer[((udBackgroundVoltageBufferIndex - 1) MOD 100) + 1];
        fBackgroundVoltageBuffer[((udBackgroundVoltageBufferIndex - 1) MOD 100) + 1] := fBackgroundVoltageAcc / uAccCount;
        // Remove overwritten voltage
        IF udBackgroundVoltageBufferIndex > 100 THEN
            fBackgroundVoltageSum := fBackgroundVoltageSum - fBackgroundVoltageStale;
        END_IF
        fBackgroundVoltageSum := fBackgroundVoltageSum + fBackgroundVoltageAcc / uAccCount;
        fBackgroundVoltageAcc := fVoltage;
        uAccCount := 1;
        udBackgroundVoltageBufferIndex := udBackgroundVoltageBufferIndex + 1;
    ELSE
        uAccCount := uAccCount + 1;
        fBackgroundVoltageAcc := fBackgroundVoltageAcc + fVoltage;
    END_IF

END_IF

IF udBackgroundVoltageBufferIndex <> 1 AND BACKGROUND_MODE = Auto THEN
    fBackgroundVoltage := fBackgroundVoltageSum / MIN((udBackgroundVoltageBufferIndex - 1), 100);
END_IF

// Start collecting background in manual mode - 60s by default but can be set with uBackgroundCollectionTime
IF bBackgroundCollect = TRUE AND BACKGROUND_MODE = Manual THEN
    bBackgroundCollect := FALSE;
    udBackgroundManualCount := 0;
    fBackgroundVoltage := 0;
    tofBackgroundCollecting(IN := TRUE);
END_IF

bBackgroundCollecting := FALSE;
tofBackgroundCollecting(IN := FALSE, PT := UINT_TO_TIME(uBackgroundCollectionTime * 1000));
IF tofBackgroundCollecting.Q = TRUE THEN
    IF BACKGROUND_MODE = Manual THEN
        bBackgroundCollecting := TRUE;
        udBackgroundManualCount := udBackgroundManualCount + 1;
        fBackgroundVoltage := (fBackgroundVoltage * (udBackgroundManualCount - 1) + fVoltage) / udBackgroundManualCount;
    END_IF
END_IF

// Getting frequency based on accelerator source
{IF defined (K)}
    IF PMPS_GVL.stCurrentBeamParameters.nMachineMode = 0 THEN
        fFrequency := fSXR_NC_Frequency;
    ELSIF PMPS_GVL.stCurrentBeamParameters.nMachineMode = 1 THEN
        fFrequency := uSXR_SC_Frequency;
    END_IF
{ELSIF defined (L)}
    IF PMPS_GVL.stCurrentBeamParameters.nMachineMode = 0 THEN
        fFrequency := fHXR_NC_Frequency;
    ELSIF PMPS_GVL.stCurrentBeamParameters.nMachineMode = 1 THEN
        fFrequency := uHXR_SC_Frequency;
    END_IF
{END_IF}

// Getting wattage and energy
fPulseWattage := SEL(fResponsivity <> 0, 0, (fVoltage - fBackgroundVoltage) / fResponsivity);
fCalibMJ := SEL(fFrequency <> 0, -9999, fPulseWattage / fFrequency);

// Buffer the full-rate Voltage, Pulse wattage, and calibrated MJ values
fbVoltageBuffer(
    bExecute := TRUE,
    fInput := fVoltage,
    arrOutput => fVoltageBuffer);
fbPulseWattageBuffer(
    bExecute := TRUE,
    fInput := fPulseWattage,
    arrOutput => fPulseWattageBuffer);
fbCalibMJBuffer(
    bExecute := TRUE,
    fInput := fCalibMJ,
    arrOutput => fCalibMJBuffer);

END_FUNCTION_BLOCK

// ---- Devices/PPM/FB_PPM_Gige.TcPOU
FUNCTION_BLOCK FB_PPM_Gige
VAR
    iIlluminatorINT AT %Q*: INT;

    {attribute 'pytmc' := '
        pv: PWR
        field: ZNAM OFF
        field: ONAM ON
    '}
    bGigePower AT %Q*: BOOL;

    {attribute 'pytmc' := '
        pv: CIL:PCT
        EGU: %
    '}
    fIlluminatorPercent: LREAL;

    fbGetIllPercent: FB_AnalogInput;
    fbSetIllPercent: FB_AnalogOutput;

    bGigeInit: BOOL := FALSE;
END_VAR

// Turn the GigE on by default
IF NOT bGigeInit THEN
    bGigePower := TRUE;
    bGigeInit := TRUE;
END_IF

// Illuminator conversion to percentage
fbSetIllPercent(
    fReal:=fIlluminatorPercent,
    fSafeMax:=100,
    fSafeMin:=0,
    iTermBits:=15,
    fTermMax:=100,
    fTermMin:=0,
    iRaw=>iIlluminatorINT);
fbGetIllPercent(
    iRaw:=iIlluminatorINT,
    iTermBits:=15,
    fTermMax:=100,
    fTermMin:=0,
    fReal=>fIlluminatorPercent);

END_FUNCTION_BLOCK

// ---- POUs/FB_XTES_Flowswitch.TcPOU
{attribute 'analysis' := '-33'}
FUNCTION_BLOCK FB_XTES_Flowswitch
VAR_OUTPUT
    {attribute 'pytmc' := '
        pv: FLOW_OK
        field: ZNAM LOW
        field: ONAM OK
    '}
    bFlowOk AT %I*: BOOL;
END_VAR

END_FUNCTION_BLOCK

// ---- Tests/FB_REFTest.TcPOU
(*
    Single integration smoke for FB_REF. Goal: prove the FB_REF wiring
    (REFERENCE TO refs, CallAfterInit / CallAfterInitStateMover / CallAfterInitPMPS
    chain, inline-init of fbStates, per-state name/fDelta defaults,
    PMPS state-key registration) still drives FB_MotionStageNC into the
    configured fPosition for a commanded state.
*)
{attribute 'analysis' := '-33'}
FUNCTION_BLOCK FB_REFTest EXTENDS FB_TestSuite
VAR
    axRef    : ARRAY[1..MotionConstants.MAX_STATE_MOTORS] OF AXIS_REF;
    fbPDS    : LCLS_Tc_DevAbs.FB_PersistentDataStorage;

    fbMotorX : FB_MotionStageNC(AxisRef := axRef[1], iPersistentDataStorage := fbPDS, sName := 'X');
    fbMotorY : FB_MotionStageNC(AxisRef := axRef[2], iPersistentDataStorage := fbPDS, sName := 'Y');

    aiMotionStage : ARRAY[1..MotionConstants.MAX_STATE_MOTORS] OF I_MotionStage := [fbMotorY];
    {attribute 'pytmc' := '
        pv: MMS
        array: 1..1 | 1..2
    '}
    astPositionState : ARRAY[1..MotionConstants.MAX_STATE_MOTORS]
                         OF ARRAY[1..GeneralConstants.MAX_STATES] OF ST_PositionState;

    fbFFHWO    : FB_HardwareFFOutput;
    fbArbiter  : FB_Arbiter(1);
    fbSubSysIO : FB_DummyArbIO;

    bEnableMotion         : BOOL;
    bEnableBeamParams     : BOOL;
    bEnablePositionLimits : BOOL;
    bReadDBNow            : BOOL;

    sDeviceName    : STRING := 'TST:REF';
    sTransitionKey : STRING := 'TST:REF-TRANSITION';

    (* Driven from the body to simulate the reader going busy then idle during cold start. *)
    bFileReaderBusy  : BOOL;
    bFileReaderError : BOOL;

    stDefault : ST_PositionState := (
        bMoveOk       := TRUE,
        bValid        := TRUE,
        bUseRawCounts := FALSE
    );

    afbStatePMPS : ARRAY[1..2] OF FB_CC_StatePMPSConfig[
        (stPositionState := astPositionState[1][E_EpicsInOut.OUT],
         stDefault       := stDefault,
         fPosition       := 10.0,
         sPmpsState      := 'TST:REF-OUT'),
        (stPositionState := astPositionState[1][E_EpicsInOut.IN],
         stDefault       := stDefault,
         fPosition       := 20.0,
         sPmpsState      := 'TST:REF-IN')
    ];

    fbREF : FB_REF(
        aiMotionStage    := aiMotionStage,
        astPositionState := astPositionState,
        fbFFHWO          := fbFFHWO,
        fbArbiter        := fbArbiter,
        sDeviceName      := sDeviceName,
        sTransitionKey   := sTransitionKey,
        bEnableBeamParams     := TRUE,
        bEnablePositionLimits := TRUE,
        bReadDBNow := FALSE,
        bFileReaderBusy       := bFileReaderBusy,
        bFileReaderError      := bFileReaderError
    );

    fbTestTimer : TON := (IN := TRUE, PT := T#60S);
    nTestStep   : INT;
    fGoal       : LREAL := 20.0;
    fTolerance  : LREAL := 2.0;
    fObserved   : LREAL;
    bFirstScan  : BOOL := TRUE;
    i	: UINT;
END_VAR

TEST(__POUNAME());

CASE nTestStep OF
    0:
        IF bFirstScan THEN
            fbMotorX.SetModeEnableLimits(
                LimBackward    := TRUE,
                LimForward     := TRUE,
                HomeEnable     := FALSE,
                BrakeMode      := E_StageBrakeMode.IF_ENABLED,
                EnableMode     := E_StageEnableMode.DURING_MOTION,
                HomeMode       := E_EpicsHomeCmd.LOW_LIMIT,
                UserEnable     := TRUE,
                HardwareEnable := TRUE
            );
           fbMotorX.SetVelocity(Velocity := 15.5);
           fbMotorX.RestoreMotionParams      := FALSE;
           fbMotorX.DoNotRestoreNcParameters := TRUE;

           fbMotorY.SetModeEnableLimits(
                LimBackward    := TRUE,
                LimForward     := TRUE,
                HomeEnable     := FALSE,
                BrakeMode      := E_StageBrakeMode.IF_ENABLED,
                EnableMode     := E_StageEnableMode.DURING_MOTION,
                HomeMode       := E_EpicsHomeCmd.LOW_LIMIT,
                UserEnable     := TRUE,
                HardwareEnable := TRUE
            );
            fbMotorY.SetVelocity(Velocity := 15.5);
            fbMotorY.RestoreMotionParams      := FALSE;
            fbMotorY.DoNotRestoreNcParameters := TRUE;

            bEnableMotion         := TRUE;
            bEnableBeamParams     := TRUE;
            bEnablePositionLimits := TRUE;
            bReadDBNow            := TRUE;
            bFileReaderBusy  := TRUE;
            bFileReaderError := FALSE;
            bFirstScan := FALSE;

        END_IF
        nTestStep      := 1;
    1:
        bFileReaderBusy  := FALSE;
        bFileReaderError := FALSE;
        nTestStep      := 2;
    2:
        (* Wait for cold-start stabilisation: PMPS DB parsed, motor
           ready to accept moves, no residual error. *)
        IF fbMotorY.stMotionStatus.bStageReady
           AND NOT fbMotorY.stMotionStatus.bError THEN
            fbREF.eEnumSet := E_EpicsInOut.IN;
            nTestStep      := 3;
        END_IF

    3:
        fObserved := fbMotorY.stMotionStatus.fActPosition;
        IF fbREF.eEnumGet = E_EpicsInOut.IN
           AND NOT fbMotorY.stMotionStatus.bMoving
           AND ABS(fObserved - fGoal) <= fTolerance THEN
            AssertTrue(
                Condition := TRUE,
                Message   := 'T01: REF reached IN within tolerance');
            nTestStep := 4;
        END_IF
END_CASE

fbPDS();
fbMotorX();
fbMotorY();

fbREF();

fbSubSysIO(LA := fbArbiter, FFO := fbFFHWO);
fbTestTimer();

IF nTestStep = 4 THEN
    TEST_FINISHED();
ELSIF fbTestTimer.Q THEN
    AssertTrue(
        Condition := FALSE,
        Message   := CONCAT(
            CONCAT(
                CONCAT('T01: timed out at step ', TO_STRING(nTestStep)),
                CONCAT(', eEnumGet=', TO_STRING(TO_UDINT(fbREF.eEnumGet)))),
            CONCAT(', fActPos=', TO_STRING(fObserved))));
    TEST_FINISHED();
END_IF

END_FUNCTION_BLOCK

// ---- Devices/REF/FB_REF.TcPOU
(* Reference laser (REF): thin ND-framework state-mover wrapper.
   Y in/out mover via FB_PositionStatePMPSND, plus a tick site for the
   laser power/dimmer (FB_REF_Laser). Caller-owned motors, stage/state
   arrays, fast-fault and arbiter are injected via FB_Init REFERENCE TO
   and forwarded to fbStates; enum bridge and toggles re-forwarded each cycle. *)
{attribute 'call_after_init'}
FUNCTION_BLOCK FB_REF
VAR_INPUT
    // Set this to a non-unknown value to request a new move.
    {attribute 'pytmc' := '
        pv: MMS:STATE:SET
        io: io
    '}
    eEnumSet : E_EpicsInOut;
    (* Run-time toggles forwarded into fbStates each cycle. PMPSND
       captures these by value in its own FB_Init, so the body
       re-writes fbStates.* every cycle to track live caller changes. *)
    fTermMax               : LREAL := 200;
END_VAR
VAR


    {attribute 'pytmc' := 'pv: LAS'}
    fbLaser : FB_REF_Laser;

    (* REFERENCE TO backing fields populated by FB_Init. *)
    {attribute 'no_copy'}
    aiMotionStage         : REFERENCE TO ARRAY[1..MotionConstants.MAX_STATE_MOTORS] OF I_MotionStage;
    {attribute 'no_copy'}
    astPositionState      : REFERENCE TO ARRAY[1..MotionConstants.MAX_STATE_MOTORS]
                                            OF ARRAY[1..GeneralConstants.MAX_STATES] OF ST_PositionState;
    {attribute 'no_copy'}
    fbFFHWO               : REFERENCE TO FB_HardwareFFOutput;
    {attribute 'no_copy'}
    fbArbiter             : REFERENCE TO FB_Arbiter;

    sDeviceName           : STRING;
    sTransitionKey        : STRING;
    bEnableMotion         : BOOL := TRUE;
    bEnableBeamParams     : BOOL;
    bEnablePositionLimits : BOOL;
    bReadDBNow            : BOOL;

    bFileReaderBusy       : REFERENCE TO BOOL;
    bFileReaderError      : REFERENCE TO BOOL;
    (* One configurator per REF state (OUT, IN). Writes the per-state
       sName and fDelta. Ticked cyclically in the body AFTER fbStates
       so its writes win over the template baseline FB_StateSetup
       applied via FB_CC_StatePMPSConfig *)
    afbStateDefaults : ARRAY[1..2] OF FB_CC_InternalStateConfig[
        (stPositionState := astPositionState[1][E_EpicsInOut.OUT],
         sName           := 'OUT',
         fDelta          := FDELTA_DEFAULT),
        (stPositionState := astPositionState[1][E_EpicsInOut.IN],
         sName           := 'IN',
         fDelta          := FDELTA_DEFAULT)
    ];
    {attribute 'pytmc' := 'pv: MMS'}
    fbStates : FB_PositionStatePMPSND(
        aiMotionStage         := aiMotionStage,
        astPositionState      := astPositionState,
        nActiveMotorCount     := 1,
        eEnumSet              := eEnumSet,
        eEnumGet              := eEnumGet,
        bEnableMotion         := bEnableMotion,
        eMotionRequestPolicy  := E_MotionRequestPolicy.INTERRUPT,
        bEnableBeamParams     := bEnableBeamParams,
        bEnablePositionLimits := bEnablePositionLimits,
        bReadDBNow            := bReadDBNow,
        bFileReaderBusy       := bFileReaderBusy,
        bFileReaderError      := bFileReaderError,
        fbFFHWO               := fbFFHWO,
        fbArbiter             := fbArbiter,
        sDeviceName           := sDeviceName,
        sTransitionKey        := sTransitionKey
    );
    i : UINT;
END_VAR
VAR_OUTPUT
    // The current position state as an enum.
    {attribute 'pytmc' := '
        pv: MMS:STATE:GET
        io: i
    '}
     eEnumGet : E_EpicsInOut;
    // The PMPS database lookup associated with the current position state.
    stDbStateParams: ST_DbStateParams;
END_VAR
VAR CONSTANT
    (* REF-wide default tolerance for state in-position detection,
       applied per-state by afbStateDefaults. *)
    FDELTA_DEFAULT : LREAL := 2;
END_VAR

IF NOT __ISVALIDREF(aiMotionStage)
   OR NOT __ISVALIDREF(astPositionState)
   OR NOT __ISVALIDREF(fbFFHWO)
   OR NOT __ISVALIDREF(fbArbiter) THEN
    RETURN;
END_IF

fbStates(stDbStateParams=> stDbStateParams);

fbLaser(fTermMax := fTermMax);

(* Auto-fired after FB_Init. fbStates' inline-init ran first and
   forwarded nil refs, so this re-supplies the now-valid refs via
   fbStates.CallAfterInitStateMover / CallAfterInitPMPS and writes the
   per-state device defaults. *)
{attribute 'call_after_init'}
METHOD CallAfterInit
VAR
    i : UINT;
END_VAR
afbStateDefaults[1].CallAfterInit(
    stPositionState := THIS^.astPositionState[1][E_EpicsInOut.OUT]
);
afbStateDefaults[2].CallAfterInit(
    stPositionState := THIS^.astPositionState[1][E_EpicsInOut.IN]
);

THIS^.fbStates.CallAfterInitStateMover(
    aiMotionStage         := aiMotionStage,
    astPositionState      := astPositionState,
    nActiveMotorCount     := 1,
    eEnumSet              := eEnumSet,
    eEnumGet              := eEnumGet,
    bEnableMotion         := bEnableMotion,
    eMotionRequestPolicy  := E_MotionRequestPolicy.INTERRUPT,
);

THIS^.fbStates.CallAfterInitPMPS(
    aiMotionStage         := aiMotionStage,
    astPositionState      := astPositionState,
    bEnableBeamParams     := bEnableBeamParams,
    bEnablePositionLimits := bEnablePositionLimits,
    bReadDBNow            := bReadDBNow,
    bFileReaderBusy       := bFileReaderBusy,
    bFileReaderError      := bFileReaderError,
    fbFFHWO               := fbFFHWO,
    fbArbiter             := fbArbiter,
    sDeviceName           := sDeviceName,
    sTransitionKey        := sTransitionKey
);
END_METHOD

//FB_Init is always available implicitly and it is used primarily for initialization.
//The return value is not evaluated. For a specific influence, you can also declare the
//methods explicitly and provide additional code there with the standard initialization
//code. You can evaluate the return value.
METHOD FB_Init: BOOL
VAR_INPUT
    bInitRetains: BOOL; // TRUE: the retain variables are initialized (reset warm / reset cold)
    bInCopyCode: BOOL;  // TRUE: the instance will be copied to the copy code afterward (online change)
    aiMotionStage          : REFERENCE TO ARRAY[1..MotionConstants.MAX_STATE_MOTORS] OF I_MotionStage;
    astPositionState       : REFERENCE TO ARRAY[1..MotionConstants.MAX_STATE_MOTORS]
                                            OF ARRAY[1..GeneralConstants.MAX_STATES] OF ST_PositionState;
    fbFFHWO                : REFERENCE TO FB_HardwareFFOutput;
    fbArbiter              : REFERENCE TO FB_Arbiter;
    sDeviceName            : STRING;
    sTransitionKey         : STRING;
    bEnableBeamParams      : BOOL;
    bEnablePositionLimits  : BOOL;
    bReadDBNow             : BOOL;
    bFileReaderBusy       : REFERENCE TO BOOL;
    bFileReaderError      : REFERENCE TO BOOL;
END_VAR
THIS^.aiMotionStage    REF= aiMotionStage;
THIS^.astPositionState REF= astPositionState;
THIS^.fbFFHWO          REF= fbFFHWO;
THIS^.fbArbiter        REF= fbArbiter;
THIS^.sDeviceName      := sDeviceName;
THIS^.sTransitionKey   := sTransitionKey;
THIS^.bEnableBeamParams    := bEnableBeamParams;
THIS^.bEnablePositionLimits:= bEnablePositionLimits;
THIS^.bReadDBNow           := bReadDBNow;
THIS^.bFileReaderBusy       REF= bFileReaderBusy;
THIS^.bFileReaderError      REF= bFileReaderError;
END_METHOD

PROPERTY MaintMode : BOOL
GET
MaintMode := fbStates.stPMPSEpicsToPlc.bMaintMode;
END_GET
SET
fbStates.stPMPSEpicsToPlc.bMaintMode := MaintMode;
END_SET
END_PROPERTY

END_FUNCTION_BLOCK

// ---- Devices/REF/FB_REF_Laser.TcPOU
FUNCTION_BLOCK FB_REF_Laser
VAR_INPUT
    {attribute 'pytmc' := '
        pv: SHUTDOWN
        io: io
    '}
    bShutdown: BOOL;

    {attribute 'pytmc' := '
        pv: PCT
        io: io
    '}
    fLaserPercent: LREAL;

    fTermMax: LREAL := 200;
END_VAR
VAR
    iShutdownINT AT %Q*: INT;
    iLaserINT AT %Q*: INT;

    fbGetLasPercent: FB_AnalogInput;
    fbSetLasPercent: FB_AnalogOutput;
END_VAR

// Send 5V to suppress laser
IF bShutdown THEN
    iShutdownINT := LREAL_TO_INT(EXPT(2, 14));
ELSE
    iShutdownINT := 0;
END_IF

// Limit to 0-5V instead of 10V
fbSetLasPercent(
    fReal:=fLaserPercent,
    fSafeMax:=100,
    fSafeMin:=0,
    iTermBits:=15,
    fTermMax:=fTermMax,
    fTermMin:=0,
    iRaw=>iLaserInt);
fbGetLasPercent(
    iRaw:=iLaserInt,
    iTermBits:=15,
    fTermMax:=fTermMax,
    fTermMin:=0,
    fReal=>fLaserPercent);

END_FUNCTION_BLOCK

// ---- Tests/FB_SATTTest.TcPOU
FUNCTION_BLOCK FB_SATTTest EXTENDS FB_TestSuite
VAR

    axRef    : AXIS_REF;
    fbPDS    : LCLS_Tc_DevAbs.FB_PersistentDataStorage;

    fbMotorY      : FB_MotionStageNC(AxisRef := axRef, iPersistentDataStorage := fbPDS, sName := 'Y');
    aiMotionStage : ARRAY[1..MotionConstants.MAX_STATE_MOTORS] OF I_MotionStage := [fbMotorY];

    {attribute 'pytmc' := '
        pv: MMS
        array: 1..1 | 1..9
    '}
    astPositionState : ARRAY[1..MotionConstants.MAX_STATE_MOTORS]
                         OF ARRAY[1..GeneralConstants.MAX_STATES] OF ST_PositionState;

    fbFFHWO : FB_HardwareFFOutput;

    sDeviceName : STRING := 'AT1K4:L2SI';
    bFileReaderBusy :  BOOL;
    fbArbiter  : FB_Arbiter(1);
    fbSubSysIO : FB_DummyArbIO;

    fbSATT : FB_SXR_SATT_Stage(
        aiMotionStage    := aiMotionStage,
        astPositionState := astPositionState,
        fbFFHWO          := fbFFHWO,
        bFileReaderBusy  := bFileReaderBusy,
        sDeviceName      := sDeviceName,
        RTDPMPSState     := 'AT1K4:L2SI-RTD'
    );

    stDefault : ST_PositionState := (
        fDelta        := 0.2,
        bMoveOk       := TRUE,
        bValid        := TRUE,
        bUseRawCounts := FALSE
    );

    afbStateDefaults : ARRAY[1..9] OF FB_CC_StateDefaultsConfig[
        (stPositionState := astPositionState[1][E_SXR_SATT_Position.OUT],     stDefault := stDefault, sName := 'Out',     fPosition := 10),
        (stPositionState := astPositionState[1][E_SXR_SATT_Position.FILTER1], stDefault := stDefault, sName := 'Filter1', fPosition := 20),
        (stPositionState := astPositionState[1][E_SXR_SATT_Position.FILTER2], stDefault := stDefault, sName := 'Filter2', fPosition := 30),
        (stPositionState := astPositionState[1][E_SXR_SATT_Position.FILTER3], stDefault := stDefault, sName := 'Filter3', fPosition := 40),
        (stPositionState := astPositionState[1][E_SXR_SATT_Position.FILTER4], stDefault := stDefault, sName := 'Filter4', fPosition := 50),
        (stPositionState := astPositionState[1][E_SXR_SATT_Position.FILTER5], stDefault := stDefault, sName := 'Filter5', fPosition := 60),
        (stPositionState := astPositionState[1][E_SXR_SATT_Position.FILTER6], stDefault := stDefault, sName := 'Filter6', fPosition := 70),
        (stPositionState := astPositionState[1][E_SXR_SATT_Position.FILTER7], stDefault := stDefault, sName := 'Filter7', fPosition := 80),
        (stPositionState := astPositionState[1][E_SXR_SATT_Position.FILTER8], stDefault := stDefault, sName := 'Filter8', fPosition := 90)
    ];

    (* Per-filter material + thickness (integrator-owned) written into
       the device's arrFilters table via FB_SATT_FilterConfig. *)
    afbFilterCfg : ARRAY[1..8] OF FB_SATT_FilterConfig[
        (stFilter := fbSATT.arrFilters[1], sFilterMaterial := 'C',  fFilterThickness_um := 25),
        (stFilter := fbSATT.arrFilters[2], sFilterMaterial := 'C',  fFilterThickness_um := 50),
        (stFilter := fbSATT.arrFilters[3], sFilterMaterial := 'C',  fFilterThickness_um := 100),
        (stFilter := fbSATT.arrFilters[4], sFilterMaterial := 'Si', fFilterThickness_um := 200),
        (stFilter := fbSATT.arrFilters[5], sFilterMaterial := 'Si', fFilterThickness_um := 320),
        (stFilter := fbSATT.arrFilters[6], sFilterMaterial := 'Si', fFilterThickness_um := 640),
        (stFilter := fbSATT.arrFilters[7], sFilterMaterial := 'Si', fFilterThickness_um := 1280),
        (stFilter := fbSATT.arrFilters[8], sFilterMaterial := 'Si', fFilterThickness_um := 2560)
    ];

    bFirstScan : BOOL := TRUE;
    i          : UINT;
END_VAR

IF bFirstScan THEN
    fbMotorY.SetModeEnableLimits(
        LimBackward    := TRUE,
        LimForward     := TRUE,
        HomeEnable     := FALSE,
        BrakeMode      := E_StageBrakeMode.NO_BRAKE,
        EnableMode     := E_StageEnableMode.DURING_MOTION,
        HomeMode       := E_EpicsHomeCmd.NONE,
        UserEnable     := TRUE,
        HardwareEnable := TRUE
    );
    fbMotorY.SetVelocity(Velocity := 15.5);
    fbMotorY.RestoreMotionParams      := FALSE;
    fbMotorY.DoNotRestoreNcParameters := TRUE;
    bFirstScan := FALSE;
END_IF
// avoid a division by Zero in F_CalculateAbsorbptionConstant from Physics Library
// protection must be added there on neV
PMPS_GVL.stCurrentBeamParameters.neV := 250.0;
fbPDS();
fbMotorY();
fbSATT();
fbSubSysIO(LA := fbArbiter, FFO := fbFFHWO);

TestConfig();
TestStateMove();
TestTempFFO();

METHOD AssertBothTempFault
VAR_INPUT
    Message : STRING;
END_VAR

AssertFalse(
    fbSATT.fbRTD_1.FFO.i_xOK,
    CONCAT('SATT RTD1 expected fault: ', Message)
);
AssertFalse(
    fbSATT.fbRTD_2.FFO.i_xOK,
    CONCAT('SATT RTD2 expected fault: ', Message)
);
END_METHOD

METHOD AssertNeitherTempFault
VAR_INPUT
    Message : STRING;
END_VAR

AssertTrue(
    fbSATT.fbRTD_1.FFO.i_xOK,
    CONCAT('SATT RTD1 expected ok: ', Message)
);
AssertTrue(
    fbSATT.fbRTD_2.FFO.i_xOK,
    CONCAT('SATT RTD2 expected ok: ', Message)
);
END_METHOD

METHOD SetSATTTemp
VAR_INPUT
    iTempC : INT;
END_VAR
VAR
    ptr : POINTER TO INT;
END_VAR

ptr  := ADR(fbSATT.fbRTD_1.iRaw);
ptr^ := iTempC * 100;

ptr  := ADR(fbSATT.fbRTD_2.iRaw);
ptr^ := iTempC * 100;
END_METHOD

(*
    Verifies the integrator-side configurators each write their own
    slot fields exactly once at init, with no overlap:
      - FB_CC_StateDefaultsConfig -> sName, fPosition, and fDelta from
        the stDefault baseline
      - FB_SATT_FilterConfig      -> arrFilters material, thickness
    All are one-shot CallAfterInit writes, so the values are present
    from the first scan; this test asserts once and finishes.
*)
METHOD TestConfig
VAR CONSTANT
    fTol : LREAL := 0.001;
END_VAR
TEST('TestSATTConfig');

(* FB_CC_StateDefaultsConfig wrote sName + the fDelta baseline. *)
AssertTrue(
    astPositionState[1][E_SXR_SATT_Position.OUT].sName = 'Out',
    'OUT sName not set by FB_CC_StateDefaultsConfig');
AssertTrue(
    ABS(astPositionState[1][E_SXR_SATT_Position.OUT].fDelta - 0.2) <= fTol,
    'OUT fDelta not copied from stDefault by FB_CC_StateDefaultsConfig');
AssertTrue(
    astPositionState[1][E_SXR_SATT_Position.FILTER1].sName = 'Filter1',
    'FILTER1 sName not set by FB_CC_StateDefaultsConfig');

(* FB_CC_StateDefaultsConfig wrote fPosition. *)
AssertTrue(
    ABS(astPositionState[1][E_SXR_SATT_Position.OUT].fPosition - 10.0) <= fTol,
    'OUT fPosition not set by FB_CC_StateDefaultsConfig');
AssertTrue(
    ABS(astPositionState[1][E_SXR_SATT_Position.FILTER1].fPosition - 20.0) <= fTol,
    'FILTER1 fPosition not set by FB_CC_StateDefaultsConfig');

(* FB_SATT_FilterConfig wrote material + thickness into arrFilters. *)
AssertTrue(
    fbSATT.arrFilters[1].sFilterMaterial = 'C',
    'arrFilters[1] material not set by FB_SATT_FilterConfig');
AssertTrue(
    ABS(fbSATT.arrFilters[1].fFilterThickness_um - 25.0) <= fTol,
    'arrFilters[1] thickness not set by FB_SATT_FilterConfig');

TEST_FINISHED();
END_METHOD

(*
    Smoke test for SATT state-move wiring. Walks OUT then FILTER1 and
    asserts each lands within fTolerance of the configured fPosition.
    Mirrors FB_REFTest: stageReady gate up front, NOT bMoving +
    position-tolerance check per state, 60s watchdog, on timeout
    AssertTrue(FALSE, ...) with the current step and observed
    position. Two moves is enough to exercise the FB wiring; the
    motion stack itself is covered by the
    lcls-twincat-motion-abstraction test suite.
*)
METHOD TestStateMove
VAR_INST
    tonTimer  : TON;
    nTestStep : INT := 0;
    fObserved : LREAL;
END_VAR
VAR CONSTANT
    fTolerance : LREAL := 2.0;
END_VAR
TEST('TestSATTStateMove');

tonTimer(IN := TRUE, PT := T#60s);
fObserved := fbMotorY.stMotionStatus.fActPosition;

CASE nTestStep OF
    0:

        IF fbMotorY.stMotionStatus.bStageReady
           AND NOT fbMotorY.stMotionStatus.bError THEN
            fbSATT.eEnumSet := E_SXR_SATT_Position.OUT;
            nTestStep       := 1;
        END_IF
    1:
        (* OUT is configured at fPosition := 10 in afbStateDefaults[1]. *)
        IF fbSATT.eEnumGet = E_SXR_SATT_Position.OUT
           AND NOT fbMotorY.stMotionStatus.bMoving
           AND ABS(fObserved - 10.0) <= fTolerance THEN
            fbSATT.eEnumSet := E_SXR_SATT_Position.FILTER1;
            nTestStep       := 2;
        END_IF
    2:
        (* FILTER1 is configured at fPosition := 20 in afbStateDefaults[2]. *)
        IF fbSATT.eEnumGet = E_SXR_SATT_Position.FILTER1
           AND NOT fbMotorY.stMotionStatus.bMoving
           AND ABS(fObserved - 20.0) <= fTolerance THEN
            AssertTrue(
                Condition := TRUE,
                Message   := 'TestSATTStateMove: OUT then FILTER1 reached within tolerance');
            nTestStep := 3;
        END_IF
END_CASE

IF nTestStep = 3 THEN
    TEST_FINISHED();
ELSIF tonTimer.Q THEN
    AssertTrue(
        Condition := FALSE,
        Message   := CONCAT(
            CONCAT(
                CONCAT('TestSATTStateMove: timed out at step ', TO_STRING(nTestStep)),
                CONCAT(', eEnumGet=', TO_STRING(TO_UDINT(fbSATT.eEnumGet)))),
            CONCAT(', fActPos=', TO_STRING(fObserved))));
    TEST_FINISHED();
END_IF
END_METHOD

METHOD TestTempFFO
VAR_INST
    tonTimer    : TON;
    nStep       : UINT := 0;
    bOutChecked : BOOL := FALSE;
    bInChecked  : BOOL := FALSE;
END_VAR
VAR CONSTANT
    nLastStep : UINT := 3;
END_VAR

(* Do we fault at the correct times?
   Parasitically depends on state move test. *)
TEST('TestSATTTempFFO');

(* Prepare a timeout *)
tonTimer(IN := TRUE, PT := T#10s);

CASE nStep OF
    0:
        (* Set the thermocouple temperatures to crazy high number. *)
        SetSATTTemp(100);
        nStep := nStep + 1;
    1:
        (* Wait till we see "OUT" state and one other state (OUT
           should be no fault). *)
        IF fbSATT.eEnumGet = E_SXR_SATT_Position.OUT THEN
            AssertNeitherTempFault('was in out position');
            bOutChecked := TRUE;
        ELSIF fbSATT.eEnumGet <> E_SXR_SATT_Position.UNKNOWN THEN
            AssertBothTempFault('was in a target position');
            bInChecked := TRUE;
        END_IF
        IF bOutChecked AND bInChecked THEN
            nStep := nStep + 1;
        END_IF
    2:
        (* Set the thermocouple temperatures to low again. *)
        SetSATTTemp(0);
        nStep := nStep + 1;
    3:
        AssertNeitherTempFault('has low temp reading');
        nStep := nStep + 1;
END_CASE

IF tonTimer.Q OR nStep > nLastStep THEN
    AssertFalse(tonTimer.Q, 'Timeout in SATT temp FFO test');
    TEST_FINISHED();
END_IF
END_METHOD

END_FUNCTION_BLOCK

// ---- Devices/SATT/FB_SXR_SATT_Stage.TcPOU
(* Single Solid Attenuator (SATT) filter stack (L2SI compact, 4 stacks
   of 8 filters): single-axis mover via FB_PositionStateND (states OUT,
   FILTER1..FILTER8). Not a PMPS state mover; only RTD reactive-temp
   fault thresholds and a "device moving" fast fault. Per-cycle transmission
   from filter material/thickness and beam energy. Deps injected via FB_Init. *)
{attribute 'call_after_init'}
FUNCTION_BLOCK FB_SXR_SATT_Stage
VAR_INPUT
    (* Callers drive moves with`fbSATT.eEnumSet := E_SXR_SATT_Position.FILTER1;`. *)
    // Set this to a non-unknown value to request a new move.
    {attribute 'pytmc' := '
        pv: STATE:SET
        io: io
    '}
    eEnumSet : E_SXR_SATT_Position;
    (* Per-filter material / thickness table. Used by the transmission
       calculation. Index 1 corresponds to FILTER1 (which is the
       state at slot 2 in astPositionState, since OUT lives at slot 1
       in E_SXR_SATT_Position). *)
    {attribute 'pytmc' := 'pv: FILTERS'}
    arrFilters : ARRAY[1..8] OF ST_SATT_Filter;
END_VAR
VAR_OUTPUT
    fTemp1                    : LREAL;
    fTemp2                    : LREAL;
    bIsStationary             : BOOL;
    bError                    : BOOL;
    // The current position state as an enum.
    {attribute 'pytmc' := '
        pv: STATE:GET
        io: i
    '}
    eEnumGet : E_SXR_SATT_Position;
    {attribute 'pytmc' := '
        pv: MATERIAL
        io: i
    '}
    sActiveFilterMaterial     : STRING;

    {attribute 'pytmc' := '
        pv: THICKNESS
        io: i
        field: EGU um
    '}
    fActiveFilterThickness_um : LREAL;

    {attribute 'pytmc' := '
        pv: TRANSMISSION
        io: i
        field: DESC Filter transmission
    '}
    fTransmission             : LREAL;
    fActiveFilterDensity      : LREAL;
    fActiveFilterAtomicMass   : LREAL;
    fAbsorptionConstant       : LREAL;

    iFilterIndex              : INT := 0;
END_VAR
VAR
    fbStates : FB_PositionStateND(
        aiMotionStage        := aiMotionStage,
        astPositionState     := astPositionState,
        nActiveMotorCount    := 1,
        eEnumSet             := eEnumSet,
        eEnumGet             := eEnumGet,
        bEnableMotion        := bEnableMotion,
        eMotionRequestPolicy := E_MotionRequestPolicy.INTERRUPT
    );

    fbAtomicMass               : FB_AtomicMass;
    fbAttenuatorElementDensity : FB_AttenuatorElementDensity;

    (* EL3202-0020: 0.01 deg C per digit. Vetoed when the stage is in
       OUT (no filter in beam, no temperature to monitor). *)
    {attribute 'pytmc' := 'pv: RTD:1'}
    fbRTD_1 : FB_CC_TempSensor := (fResolution := 0.01);
    {attribute 'pytmc' := 'pv: RTD:2'}
    fbRTD_2 : FB_CC_TempSensor := (fResolution := 0.01);

    bFileReaderBusy       : REFERENCE TO BOOL;
    (* Per-cycle JSON DB read for the currently active filter's
       PMPS state, just to pull the reactive temp setpoint into
       astPickedDB[1].stReactiveParams.nTempSP. Not a PMPS BPTM
       participant; just borrows the DB pipeline. *)
    fbReadPMPSDB : FB_JsonDocToSafeBP;
    astPickedDB  : ARRAY[1..1] OF ST_DbStateParams;

    (* "Device is moving" fast fault. Raised while the Y motor is
       moving or while we are sitting in UNKNOWN. *)
    fbFF : FB_FastFault := (
        i_Desc       := 'Device is moving',
        i_TypeCode   := E_MotionFFType.DEVICE_MOVE,
        i_xAutoReset := TRUE
    );

    (* REFERENCE TO backing fields populated by FB_Init. *)
    {attribute 'no_copy'}
    aiMotionStage    : REFERENCE TO ARRAY[1..MotionConstants.MAX_STATE_MOTORS] OF I_MotionStage;
    {attribute 'no_copy'}
    astPositionState : REFERENCE TO ARRAY[1..MotionConstants.MAX_STATE_MOTORS]
                                          OF ARRAY[1..GeneralConstants.MAX_STATES] OF ST_PositionState;
    {attribute 'no_copy'}
    fbFFHWO          : REFERENCE TO FB_HardwareFFOutput;
    sDeviceName      : STRING;
    (* PMPS DB key for the RTD reactive-temperature read. The filters are not real PMPS states,
        so this device-level key names the DB entry to pull the reactive temp setpoint from.
    *)
    RTDPMPSState     : STRING;
    bEnableMotion    : BOOL := TRUE;
END_VAR

(* Nil-ref guards: every REFERENCE TO backing field must be bound. *)
IF NOT __ISVALIDREF(aiMotionStage)
   OR NOT __ISVALIDREF(astPositionState)
   OR NOT __ISVALIDREF(fbFFHWO) THEN
    RETURN;
END_IF

fbStates();

(* Filter index is offset by one because E_SXR_SATT_Position.OUT
   occupies slot 1 and FILTER1..FILTER8 occupy slots 2..9. *)
iFilterIndex := UINT_TO_INT(eEnumGet) - 1;

IF iFilterIndex >= 1 AND iFilterIndex <= 8 THEN
    sActiveFilterMaterial     := arrFilters[iFilterIndex].sFilterMaterial;
    fActiveFilterThickness_um := arrFilters[iFilterIndex].fFilterThickness_um;

    fbAtomicMass(
        sName  := sActiveFilterMaterial,
        fValue => fActiveFilterAtomicMass
    );
    fbAttenuatorElementDensity(
        sName    := sActiveFilterMaterial,
        fDensity => fActiveFilterDensity
    );

    fAbsorptionConstant := F_CalculateAbsorptionConstant(
        sElement      := sActiveFilterMaterial,
        fEnergyEV     := PMPS_GVL.stCurrentBeamParameters.neV,
        fDensity_gm3  := fActiveFilterDensity,
        fAtomicWeight := fActiveFilterAtomicMass,
        bError        => bError
    );
    fTransmission := F_CalculateTransmission(
        fAbsorptionConstant := fAbsorptionConstant,
        fThickness_in_m     := fActiveFilterThickness_um * 1.0E-6
    );
ELSE
    sActiveFilterMaterial     := '';
    fActiveFilterThickness_um := 0.0;
    fAbsorptionConstant       := 0.0;
    fActiveFilterDensity      := 0.0;
    fActiveFilterAtomicMass   := 0.0;
    fTransmission             := 1.0;
END_IF

(* "Device is moving" fault: stationary AND known position. Reads the
   motor's NC status through the I_MotionStage interface; aiMotionStage
   was nil-guarded above so slot 1 deref is safe. *)
bIsStationary := NOT aiMotionStage[1].Axis.Status.Moving;
fbFF(
    i_DevName  := sDeviceName,
    i_xOK      := bIsStationary AND eEnumGet <> E_SXR_SATT_Position.UNKNOWN,
    io_fbFFHWO := fbFFHWO
);

(* The RTD reactive-temperature read is keyed on the device-level
   RTDPMPSState (the filters are not real PMPS states, so no per-
   filter key is scanned). The named DB entry must exist; the
   temperature field may be blank. *)
astPickedDB[1].sPmpsState := RTDPMPSState;

fbReadPMPSDB(
    bExecute    := NOT bFileReaderBusy,
    jsonDoc     := PMPS_GVL.BP_jsonDoc,
    sDeviceName := sDeviceName,
    arrStates   := astPickedDB,
    io_fbFFHWO  := fbFFHWO
);

fbRTD_1(
    fFaultThreshold := astPickedDB[1].stReactiveParams.nTempSP,
    sDevName        := sDeviceName,
    bVeto           := eEnumGet = E_SXR_SATT_Position.OUT,
    io_fbFFHWO      := fbFFHWO
);
fTemp1 := fbRTD_1.fTemp;

fbRTD_2(
    fFaultThreshold := astPickedDB[1].stReactiveParams.nTempSP,
    sDevName        := sDeviceName,
    bVeto           := eEnumGet = E_SXR_SATT_Position.OUT,
    io_fbFFHWO      := fbFFHWO
);
fTemp2 := fbRTD_2.fTemp;

(* Auto-fired after FB_Init. fbStates' inline-init ran first and
   forwarded nil refs, so this re-supplies the now-valid refs via
   fbStates.CallAfterInitStateMover, running the Core / ND wiring chain. *)
{attribute 'call_after_init'}
METHOD CallAfterInit
THIS^.fbStates.CallAfterInitStateMover(
    aiMotionStage         := aiMotionStage,
    astPositionState      := astPositionState,
    nActiveMotorCount     := 1,
    eEnumSet              := eEnumSet,
    eEnumGet              := eEnumGet,
    bEnableMotion         := bEnableMotion,
    eMotionRequestPolicy  := E_MotionRequestPolicy.INTERRUPT,
);
END_METHOD

(* Stores all FB_Init inputs into instance fields. Every input is
   REFERENCE TO and is REF= bound for the lifetime of the FB.
   Inline-init of fbStates above runs first, capturing the FB_Init
   params at construction time; this method then records the same
   references on THIS^ for body-side use and live caller writes. *)
{attribute 'analysis' := '-33'}
METHOD FB_Init : BOOL
VAR_INPUT
    bInitRetains     : BOOL;
    bInCopyCode      : BOOL;
    aiMotionStage    : REFERENCE TO ARRAY[1..MotionConstants.MAX_STATE_MOTORS] OF I_MotionStage;
    astPositionState : REFERENCE TO ARRAY[1..MotionConstants.MAX_STATE_MOTORS]
                                          OF ARRAY[1..GeneralConstants.MAX_STATES] OF ST_PositionState;
    bFileReaderBusy       : REFERENCE TO BOOL;
    fbFFHWO          : REFERENCE TO FB_HardwareFFOutput;
    sDeviceName      : STRING;
    RTDPMPSState     : STRING;
END_VAR
THIS^.aiMotionStage    REF= aiMotionStage;
THIS^.astPositionState REF= astPositionState;
THIS^.fbFFHWO          REF= fbFFHWO;
THIS^.bFileReaderBusy 	REF=bFileReaderBusy;
THIS^.sDeviceName      := sDeviceName;
THIS^.RTDPMPSState     := RTDPMPSState;
END_METHOD

END_FUNCTION_BLOCK

// ---- Devices/SATT/FB_AttenuatorElementDensity.TcPOU
FUNCTION_BLOCK FB_AttenuatorElementDensity
VAR_INPUT
    sName : STRING;
END_VAR
VAR_OUTPUT
    fDensity : LREAL;
END_VAR
VAR
    fbElementDensity : FB_ElementDensity;
END_VAR

IF sName = 'C' THEN
    (* Special-case diamond here *)
    fDensity := 3.51E6;  (* C (Diamond) g/m^3 *)
ELSE
    fbElementDensity(sName:=sName);
    IF fbElementDensity.bFound THEN
        fDensity := fbElementDensity.fValue * 1.0E6; (* g/cm^3 -> g/m^3 *)
    ELSE
        fDensity := 0.0;
    END_IF
END_IF

END_FUNCTION_BLOCK

// ---- POUs/FB_CC_StateDefaultsConfig.TcPOU
(*
    Integrator-side, auto-fired writer of a complete ST_PositionState
    slot for devices whose states are not PMPS states. Functionally
    FB_CC_StatePMPSConfig without sPmpsState: copies the shared
    baseline (bMoveOk, bValid, bUseRawCounts, bLocked, nEncoderCount,
    fDelta) from the caller's stDefault template, then overlays the
    per-state sName and fPosition.

    Use this when the integrator owns the full state config and the
    device has no per-state PMPS key (e.g. FB_SXR_SATT_Stage). One
    instance per state; with this FB the integrator needs no separate
    FB_CC_StatePMPSConfig.

    Driven by {attribute 'call_after_init'}, so it is declared inline
    in the integrator box with no explicit call. The inner
    FB_StateSetup is wired at init purely as a defensive backstop, so
    a stray cyclic call stays safe and template-aware.

    One-shot write from CallAfterInit; the body is empty, so
    online-view edits to the slot persist.

    Usage (integrator declaration box):
        afbStates : ARRAY[1..N] OF FB_CC_StateDefaultsConfig[
            (stPositionState := astPositionState[1][E_xxx.OUT],
             stDefault       := stDefault,
             sName           := 'Out',
             fPosition       := 22.70),
            ...];
*)
{attribute 'call_after_init'}
FUNCTION_BLOCK FB_CC_StateDefaultsConfig
VAR_INPUT
END_VAR
VAR
    {attribute 'no_copy'}
    stPositionState : REFERENCE TO ST_PositionState;
    {attribute 'no_copy'}
    stDefault       : REFERENCE TO ST_PositionState;
    sName           : STRING;
    fPosition       : LREAL;
    fbStateSetup    : FB_StateSetup(
        stDefault       := stDefault,
        stPositionState := stPositionState,
        bSetDefault     := TRUE
    );
END_VAR

(* Re-binds the inner FB_StateSetup's REFs after FB_Init (defensive),
   then performs a one-shot write of the slot: shared baseline
   (including fDelta) from stDefault, then the per-state sName /
   fPosition overlay. No sPmpsState. Auto-fired by the runtime after
   FB_Init. *)
{attribute 'call_after_init'}
METHOD CallAfterInit
VAR_INPUT
END_VAR
THIS^.fbStateSetup.CallAfterInit(
    stDefault       := THIS^.stDefault,
    stPositionState := THIS^.stPositionState,
    bSetDefault     := TRUE
);

IF __ISVALIDREF(THIS^.stPositionState) AND __ISVALIDREF(THIS^.stDefault) THEN
    THIS^.stPositionState.bMoveOk       := THIS^.stDefault.bMoveOk;
    THIS^.stPositionState.bValid        := THIS^.stDefault.bValid;
    THIS^.stPositionState.bUseRawCounts := THIS^.stDefault.bUseRawCounts;
    THIS^.stPositionState.bLocked       := THIS^.stDefault.bLocked;
    THIS^.stPositionState.nEncoderCount := THIS^.stDefault.nEncoderCount;
    THIS^.stPositionState.fDelta        := THIS^.stDefault.fDelta;

    THIS^.stPositionState.sName     := THIS^.sName;
    THIS^.stPositionState.fPosition := THIS^.fPosition;
END_IF
END_METHOD

(* Stores the slot reference, the device-common stDefault template
   REF, plus the per-state sName / fPosition at instantiation. *)
METHOD FB_Init : BOOL
VAR_INPUT
    bInitRetains    : BOOL;
    bInCopyCode     : BOOL;
    stPositionState : REFERENCE TO ST_PositionState;
    stDefault       : REFERENCE TO ST_PositionState;
    sName           : STRING;
    fPosition       : LREAL;
END_VAR
THIS^.stPositionState REF= stPositionState;
THIS^.stDefault       REF= stDefault;
THIS^.sName            := sName;
THIS^.fPosition        := fPosition;
END_METHOD

END_FUNCTION_BLOCK

// ---- Devices/SATT/FB_SATT_FilterConfig.TcPOU
(* Per-filter writer of one ST_SATT_Filter slot in a SATT stage's
   arrFilters table. Integrator-owned, one instance per populated slot.
   Mirrors FB_CC_StatePMPSConfig: a one-shot write of sFilterMaterial and
   fFilterThickness_um from CallAfterInit; empty body, so online edits
   persist. Slot ref and values injected via FB_Init REFERENCE TO. *)
{attribute 'call_after_init'}
FUNCTION_BLOCK FB_SATT_FilterConfig
VAR_INPUT
END_VAR
VAR
    {attribute 'no_copy'}
    stFilter            : REFERENCE TO ST_SATT_Filter;
    sFilterMaterial     : STRING;
    fFilterThickness_um : LREAL;
END_VAR

(* One-shot write of the per-filter material and thickness into the
   referenced arrFilters slot. *)
{attribute 'call_after_init'}
METHOD CallAfterInit
VAR_INPUT
END_VAR
IF __ISVALIDREF(THIS^.stFilter) THEN
    THIS^.stFilter.sFilterMaterial     := THIS^.sFilterMaterial;
    THIS^.stFilter.fFilterThickness_um := THIS^.fFilterThickness_um;
END_IF
END_METHOD

(* Stores the slot reference plus the per-filter material and
   thickness at instantiation. *)
METHOD FB_Init : BOOL
VAR_INPUT
    bInitRetains        : BOOL;
    bInCopyCode         : BOOL;
    stFilter            : REFERENCE TO ST_SATT_Filter;
    sFilterMaterial     : STRING;
    fFilterThickness_um : LREAL;
END_VAR
THIS^.stFilter REF= stFilter;
THIS^.sFilterMaterial     := sFilterMaterial;
THIS^.fFilterThickness_um := fFilterThickness_um;
END_METHOD

END_FUNCTION_BLOCK

// ---- Tests/FB_SLITS_POWERTest.TcPOU
FUNCTION_BLOCK FB_SLITS_POWERTest EXTENDS FB_TestSuite
VAR
    (* Caller-owned AxisRefs and persistent storage. In a real PRG the
       AxisRefs come from MAIN.Mxx. Indexed by E_SlitsBlade (1..4). *)
    axRef : ARRAY[1..4] OF AXIS_REF;

    fbPDS : LCLS_Tc_DevAbs.FB_PersistentDataStorage;

    (* Four blade motors, indexed by E_SlitsBlade. *)
    afbMotor : ARRAY[1..4] OF FB_MotionStageNC[
        (AxisRef := axRef[E_SlitsBlade.TOP],    iPersistentDataStorage := fbPDS, sName := 'Top'),
        (AxisRef := axRef[E_SlitsBlade.BOTTOM], iPersistentDataStorage := fbPDS, sName := 'Bottom'),
        (AxisRef := axRef[E_SlitsBlade.NORTH],  iPersistentDataStorage := fbPDS, sName := 'North'),
        (AxisRef := axRef[E_SlitsBlade.SOUTH],  iPersistentDataStorage := fbPDS, sName := 'South')
    ];

    (* I_MotionStage array bound into FB_SLITS / FB_SLITS_POWER via
       FB_Init. Order matches E_SlitsBlade (TOP / BOTTOM / NORTH /
       SOUTH = 1..4). *)
    aiMotionStage : ARRAY[1..4] OF I_MotionStage := [
        afbMotor[E_SlitsBlade.TOP],
        afbMotor[E_SlitsBlade.BOTTOM],
        afbMotor[E_SlitsBlade.NORTH],
        afbMotor[E_SlitsBlade.SOUTH]
    ];

    fbFFHWO     : FB_HardwareFFOutput;

    fbSlitsPower : FB_SLITS_POWER(
        aiMotionStage   := aiMotionStage,
        fbFFHWO         := fbFFHWO,
        sDeviceName     := 'SL1L0:POWER',
        sPmpsState      := 'SL1L0:POWER-RTD',
        bFileReaderBusy := bSimFileReaderBusy,
        fApertureMargin := 0.01 // -> must be provided here
    );

    nBlade     : INT;
    bFirstScan : BOOL := TRUE;
    bStageReady : BOOL;
    bSimFileReaderBusy : BOOL;
END_VAR

TestTempFFO();
TestApertureMotion();
fbSlitsPower(bMoveOk := TRUE);

METHOD AssertAllTempFault
VAR_INPUT
    Message : STRING;
END_VAR
AssertFalse(
    fbSlitsPower.RTD_TOP_1.FFO.i_xOK,
    CONCAT('Slits Top 1 RTD expected fault: ', Message)
);
AssertFalse(
    fbSlitsPower.RTD_TOP_2.FFO.i_xOK,
    CONCAT('Slits Top 2 RTD expected fault: ', Message)
);
AssertFalse(
    fbSlitsPower.RTD_Bottom_1.FFO.i_xOK,
    CONCAT('Slits Bottom 1 RTD expected fault: ', Message)
);
AssertFalse(
    fbSlitsPower.RTD_Bottom_2.FFO.i_xOK,
    CONCAT('Slits Bottom 2 RTD expected fault: ', Message)
);
AssertFalse(
    fbSlitsPower.RTD_North_1.FFO.i_xOK,
    CONCAT('Slits North 1 RTD expected fault: ', Message)
);
AssertFalse(
    fbSlitsPower.RTD_North_2.FFO.i_xOK,
    CONCAT('Slits North 2 RTD expected fault: ', Message)
);
AssertFalse(
    fbSlitsPower.RTD_South_1.FFO.i_xOK,
    CONCAT('Slits South 1 RTD expected fault: ', Message)
);
AssertFalse(
    fbSlitsPower.RTD_South_2.FFO.i_xOK,
    CONCAT('Slits South 2 RTD expected fault: ', Message)
);
END_METHOD

METHOD AssertNoneTempFault
VAR_INPUT
    Message : STRING;
END_VAR
AssertTrue(
    fbSlitsPower.RTD_TOP_1.FFO.i_xOK,
    CONCAT('Slits Top 1 RTD expected ok: ', Message)
);
AssertTrue(
    fbSlitsPower.RTD_TOP_2.FFO.i_xOK,
    CONCAT('Slits Top 2 RTD expected ok: ', Message)
);
AssertTrue(
    fbSlitsPower.RTD_Bottom_1.FFO.i_xOK,
    CONCAT('Slits Bottom 1 RTD expected ok: ', Message)
);
AssertTrue(
    fbSlitsPower.RTD_Bottom_2.FFO.i_xOK,
    CONCAT('Slits Bottom 2 RTD expected ok: ', Message)
);
AssertTrue(
    fbSlitsPower.RTD_North_1.FFO.i_xOK,
    CONCAT('Slits North 1 RTD expected ok: ', Message)
);
AssertTrue(
    fbSlitsPower.RTD_North_2.FFO.i_xOK,
    CONCAT('Slits North 2 RTD expected ok: ', Message)
);
AssertTrue(
    fbSlitsPower.RTD_South_1.FFO.i_xOK,
    CONCAT('Slits South 1 RTD expected ok: ', Message)
);
AssertTrue(
    fbSlitsPower.RTD_South_2.FFO.i_xOK,
    CONCAT('Slits South 2 RTD expected ok: ', Message)
);
END_METHOD

METHOD SetSlitsTemp
VAR_INPUT
    iTempC : INT;
END_VAR
VAR
    ptr : POINTER TO INT;
END_VAR
ptr  := ADR(fbSlitsPower.RTD_TOP_1.iRaw);
ptr^ := iTempC * 10;

ptr  := ADR(fbSlitsPower.RTD_TOP_2.iRaw);
ptr^ := iTempC * 10;

ptr  := ADR(fbSlitsPower.RTD_Bottom_1.iRaw);
ptr^ := iTempC * 10;

ptr  := ADR(fbSlitsPower.RTD_Bottom_2.iRaw);
ptr^ := iTempC * 10;

ptr  := ADR(fbSlitsPower.RTD_North_1.iRaw);
ptr^ := iTempC * 10;

ptr  := ADR(fbSlitsPower.RTD_North_2.iRaw);
ptr^ := iTempC * 10;

ptr  := ADR(fbSlitsPower.RTD_South_1.iRaw);
ptr^ := iTempC * 10;

ptr  := ADR(fbSlitsPower.RTD_South_2.iRaw);
ptr^ := iTempC * 10;
END_METHOD

(*
    End-to-end motion coverage against the linked NC simulation axes. An
    EPICS aperture request must flow through M_CalculatePositions ->
    M_Motion -> the blade FB_StatePTPMove movers, dispatch an absolute
    move to each blade stage, and drive each NC axis to its target. The
    test waits for every blade's actual NC position to settle on the
    aperture-math target, so it confirms the request produced real
    motion, not just a software command. Requires the four axRef entries
    to be linked to their NC axes (Axis_Slit_Top / _Bottom / _North /
    _South); without the link an axis latches bError and never moves.
*)
METHOD TestApertureMotion
VAR_INST
    tonTimer : TON;
    nStep    : UINT := 0;
END_VAR
VAR CONSTANT
    nLastStep : UINT := 1;
    fDelta    : LREAL := 0.05;
END_VAR
// Does an aperture request actually drive every blade NC axis to target?
TEST('TestSlitsApertureMotion');

tonTimer(IN := TRUE, PT := T#40S);

CASE nStep OF
    0:
        IF bFirstScan THEN
            FOR nBlade := 1 TO 4 DO
                afbMotor[nBlade].SetModeEnableLimits(
                    LimBackward    := TRUE,
                    LimForward     := TRUE,
                    HomeEnable     := FALSE,
                    BrakeMode      := E_StageBrakeMode.NO_BRAKE,
                    EnableMode     := E_StageEnableMode.DURING_MOTION,
                    HomeMode       := E_EpicsHomeCmd.NONE,
                    UserEnable     := TRUE,
                    HardwareEnable := TRUE
                );
                afbMotor[nBlade].SetMotionParam(Velocity := 15.5, Acceleration := 100, Deceleration := 100, Jerk := 1000);
                afbMotor[nBlade].RestoreMotionParams      := FALSE;
                afbMotor[nBlade].DoNotRestoreNcParameters := TRUE;
            END_FOR
            bFirstScan := FALSE;
            nStep := nStep + 1;
        END_IF
    1:
        // Per-blade encoder offsets and an aperture request inside the
        // PMPS-authorized envelope (so each axis request is accepted and
        // dispatched to the linked NC axis).


        IF bStageReady THEN
            fbSlitsPower.SetAptWidthHeight(Width:=100.0, Height:=100.0);
            fbSlitsPower.rEncoderOffsetTop    := 16.1;
            fbSlitsPower.rEncoderOffsetBottom := -11.65;
            fbSlitsPower.rEncoderOffsetNorth  := 12.45;
            fbSlitsPower.rEncoderOffsetSouth  := -16.45;
            fbSlitsPower.SetApertureRequest(ApertureSizeX := 4, ApertureSizeY := 6, CenterX := 1, CenterY := 2);
            nStep := nStep + 1;
        END_IF

    2:
        // Wait for every NC axis to reach its target:
        //   Top    =  Ygap/2 + (Ycen + offTop)    =  3 +  18.1  =  21.1
        //   Bottom = -Ygap/2 + (Ycen + offBottom) = -3 + (-9.65) = -12.65
        //   North  =  Xgap/2 + (Xcen + offNorth)  =  2 +  13.45 =  15.45
        //   South  = -Xgap/2 + (Xcen + offSouth)  = -2 + (-15.45) = -17.45
        IF ABS(afbMotor[E_SlitsBlade.TOP].MotionStatus.fActPosition    -   21.1) < fDelta
        AND ABS(afbMotor[E_SlitsBlade.BOTTOM].MotionStatus.fActPosition - (-12.65)) < fDelta
        AND ABS(afbMotor[E_SlitsBlade.NORTH].MotionStatus.fActPosition  -   15.45) < fDelta
        AND ABS(afbMotor[E_SlitsBlade.SOUTH].MotionStatus.fActPosition  - (-17.45)) < fDelta THEN
            AssertTrue(TRUE, 'All blades reached aperture target');
            nStep := nStep + 1;
        END_IF
END_CASE


fbPDS();
FOR nBlade := 1 TO 4 DO
    afbMotor[nBlade]();
    bStageReady := afbMotor[nBlade].stMotionStatus.bStageReady;
END_FOR


IF tonTimer.Q OR nStep = 3 THEN
    TEST_FINISHED();
END_IF
END_METHOD

METHOD TestTempFFO
VAR_INST
    tonTimer : TON;
    nStep    : UINT := 0;
END_VAR
VAR CONSTANT
    nLastStep : UINT := 4;
END_VAR
// Do we fault at the correct times?
TEST('TestSlitsTempFFO');

// Prepare a timeout
tonTimer(IN := TRUE, PT := T#10s);

CASE nStep OF
    0:
        // Toggle the simulated file-reader busy each cycle so fbReadPMPSDB
        // keeps seeing the rising edge (NOT bBusy) a real file read gives,
        // then hold until the resolved DB threshold appears.
        bSimFileReaderBusy := TRUE;
         nStep := nStep + 1;

    1:
        bSimFileReaderBusy :=FALSE;
        IF fbSlitsPower.RTD_TOP_1.fFaultThreshold > 0 THEN
            nStep := nStep + 1;
        END_IF
    2:
        // Set the thermocouple temperatures to a crazy-high number.
        SetSlitsTemp(100);
        nStep := nStep + 1;
    3:
        // We should see faults on all RTDs at 100C.
        AssertAllTempFault('has high temp reading');
        nStep := nStep + 1;
    4:
        // Set the thermocouple temperatures back to low.
        SetSlitsTemp(0);
        nStep := nStep + 1;
    5:
        AssertNoneTempFault('has low temp reading');
        nStep := nStep + 1;
END_CASE

IF nStep = 6 THEN
    TEST_FINISHED();
ELSIF tonTimer.Q THEN
    AssertFalse(tonTimer.Q, 'Timeout in Slits temp FFO test');
    TEST_FINISHED();
END_IF
END_METHOD

END_FUNCTION_BLOCK

// ---- Devices/SLITS/FB_SLITS_POWER.TcPOU
(* PMPS-aware (power-class) variant of FB_SLITS. Adds 8 thermocouple RTDs,
   a flow switch, a reactive-temp DB lookup (FB_JsonDocToSafeBP keyed by
   sPmpsState) driving every RTD fault, an xPMPSMode toggle, and M_UpdatePMPS.
   EXTENDS FB_SLITS; body calls SUPER^() for edge-trigger consumption then
   drives M_CalculatePositions / M_Motion behind a REF nil-guard. *)
{attribute 'analysis' := '-33'}
{attribute 'call_after_init'}
FUNCTION_BLOCK FB_SLITS_POWER EXTENDS FB_SLITS

VAR
    {attribute 'pytmc' := '
    pv: MODE
    field: ZNAM Local
    field: ONAM PMPS
    io: io
    '}
    xPMPSMode : BOOL := TRUE;

    {attribute 'pytmc' := 'pv: FSW'}
    fbFlowSwitch : FB_XTES_Flowswitch;

